// SIMATIC S7-200 project (STEP 7-Micro/WIN), CPU 224 REL 02.00

SYMBOL_TABLE Panel
LimInf_FallaCad  VD1920   // Limite inferior para falla sincronización de cadena
LimSup_FallaCad  VD1930   // Limite superior para falla sincronización de cadena
Time_Pusher_Fuera_Pos T105     // Timer, pusher fuera de posición
dAux40           VD2040   // DWAux40
dAux30           VD2030   // DWAux30
dAux20           VD2020   // DWAux20
dwAuxAlaPre      VD2004   // Aux de Alarma Presente
dwAuxMem         VD2002   // Aux Mem de Alarmas
dwAux3           VD2006   // AuxRecAlarmas
WFallas          VW100    // Para Panel_Word de Fallas en el programa
Panel_Habilitador V100.0   // Para Panel_Mark Habilitador de secuencia
Panel_Parada_Emergen V100.1   // Para Panel_Mark Parada de Emergencia (Puertas, pulsador)
Panel_Termicas1  V100.2   // Para Panel_Mark Termicas1 (Mot.Ppal, Bba Vacio, Hotmelt)
Panel_Termicas2  V100.3   // Para Panel_Mark  Termicas2 (Brazo, Pusher, Cinta Transporta.)
Panel_Cadena_Ppal V100.4   // Para Panel_Mark Seguridad Cadena principal Cortada
Panel_NO_Hay_Cajas V100.5   // Para Panel_Mark No Hay Cajas en el Cargador
Panel_Falla_MotorPusher V100.6   // Para Panel_Falla Motor Pusher
Panel_Falla_SsrPusher V100.7   // Para Panel_Falla Piston Pusher
Panel_Hotmelt_No_listo V101.0   // Para Panel_Mark Hotmelt No listo (señal externa)
Panel_Hotmelt_OFF V101.1   // Para Panel_Mark Hotmelt OFF
Panel_Cajas_Trabadas V101.2   // Para Panel_Mark Cajas Trabadas
Panel_Solapa_Trasea V101.3   // Para Panel_Mark Solapa Trasera abierta
Panel_Tiem_Sin_Hotmelt V101.4   // Para Panel_Falla por tiempo transcurrido sin Hotmelt OK
Panel_Solapa_Abierta V101.5   // Para Panel_SOLAPA TRASERA ABIERTA
Panel_Caja_Trabada_Sali V101.6   // Para Panel_CAJA NO SALIÓ DE LA MÁQUINA
Panel_FallaCajaCaida V101.7   // Para Panel_Falla caja cerrada en cadena
Panel_Falla_1SnsPucher V1836.0  // Falla Falto Confirmacion de 1 Sns del lo extremos Pusher
Panel_Falla_SsrEncDes V1836.1  // Falla SENSOR ENCOLADO DESENFOCADO
Panel_Falla_CadenaDesi V1836.2  // Falla CADENA DESINCRONIZADA
Panel_Falla_Push_Fuera V1836.3  // Falla PUSHER FUERA DE POSICION
Panel_Fall_Res_1836_4 V1836.4
Panel_Fall_Res_1836_5 V1836.5
Panel_Fall_Res_1836_6 V1836.6
Panel_Fall_Res_1836_7 V1836.7
Panel_Fall_Res_1837_0 V1837.0
Panel_Fall_Res_1837_1 V1837.1
Panel_Fall_Res_1837_2 V1837.2
Panel_Fall_Res_1837_3 V1837.3
Panel_Fall_Res_1837_4 V1837.4
Panel_Fall_Res_1837_5 V1837.5
Panel_Fall_Res_1837_6 V1837.6
Panel_Fall_Res_1837_7 V1837.7
Mem_Habilitador  V1820.0  // Memorizadas_Mark Habilitador de secuencia
Mem_Parada_Emergen V1820.1  // Memorizadas_Mark Parada de Emergencia (Puertas, pulsador)
Mem_Trmicas1     V1820.2  // Memorizadas_Mark Termicas1 (Mot.Ppal, Bba Vacio, Hotmelt)
Mem_Termicas2    V1820.3  // Memorizadas_Mark  Termicas2 (Brazo, Pusher, Cinta Transporta.)
Mem_Cadena_Ppal  V1820.4  // Memorizadas_Mark Seguridad Cadena principal Cortada
Mem_NO_Hay_Cajas V1820.5  // Memorizadas_Mark No Hay Cajas en el Cargador
Mem_Falla_MotPusher V1820.6  // Memorizadas_Falla Motor Pusher
Mem_Falla_PistPusher V1820.7  // Memorizadas_Falla Piston Pusher
Mem_Hotmelt_No_listo V1821.0  // Memorizadas_Mark Hotmelt No listo (señal externa)
Mem_Hotmelt_OFF  V1821.1  // Memorizadas_Mark Hotmelt OFF
Mem_Cajas_Trabadas V1821.2  // Memorizadas_Mark Cajas Trabadas
Mem_Solapa_Trasea V1821.3  // Memorizadas_Mark Solapa Trasera abierta
Mem_Tiem_Sin_Hotmelt V1821.4  // Memorizadas_Falla por tiempo transcurrido sin Hotmelt OK
Mem_Reserv_101_5 V1821.5  // Memorizadas_v1821.5 RESERVA
Mem_Reserv_101_6 V1821.6  // Memorizadas_v1821.6 RESERVA
Mem_Reserv_101_7 V1821.7  // Memorizadas_v1821.7 RESERVA
Tiempo_Encolado_1 VW102    // Word de tiempo para ENCOLADO 1º Solapa
Tiempo_Encolado_2 VW104    // Word de tiempo para ENCOLADO 2º Solapa
Tiempo_NO_Encolar VW106    // Word de tiempo para NO ENCOLADO
Panel_Timer_Corte_Vacio VW108    // De Panel_Word de tiempo para cortar VACIO
Panel_Sel_Caja   VW110    // De Panel Selección de Programa por Tipo de Caja
Valor_Encoder_ParaPanel VD120    // Valor Actual del Encoder al Panel
Byte_Motor_Ppal_Panel MB5      // Byte para dar marcha al motor Ppal desde el Panel
Marcha_Motor_Ppal_Panel M5.0     // Mark para dar marcha al motor Ppal desde el Panel
Panel_Tie_Enc_1_0 VW160    // Tiempo Encolado 1º Solapa Caja 15x1000
Panel_Tie_Enc_2_0 VW162    // Tiempo Encolado 2º Solapa Caja 15x1000
Panel_Tie_NoEnc_0 VW164    // Tiempo No Encolado Caja 15x1000
Panel_Tie_Enc_1_1 VW166    // Tiempo Encolado 1º Solapa Caja 12x1500
Panel_Tie_Enc_2_1 VW168    // Tiempo Encolado 2º Solapa Caja 12x1500
Panel_Tie_NoEnc_1 VW170    // Tiempo No Encolado Caja 12x1500
Panel_Tie_Enc_1_2 VW172    // Tiempo Encolado 1º Solapa Caja 12x1000
Panel_Tie_Enc_2_2 VW174    // Tiempo Encolado 2º Solapa Caja 12x1000
Panel_Tie_NoEnc_2 VW176    // Tiempo No Encolado Caja 12x1000
Panel_Tie_Enc_1_3 VW178    // Tiempo Encolado 1º Solapa Caja 12x750
Panel_Tie_Enc_2_3 VW180    // Tiempo Encolado 2º Solapa Caja 12x750
Panel_Tie_NoEnc_3 VW182    // Tiempo No Encolado Caja 12x750
Hab_Falla_18362  M29.2    // Hab_Falla_Sic_Cadena
END_SYMBOL_TABLE

SYMBOL_TABLE I/O
iEncoder_Fase_A  I0.0     // Encoder pulso A
iEncoder_Fase_B  I0.1     // Encoder pulso B
iEncoder_Cero    I0.2     // Encoder pulso 0
iSsr_Area_Encolado I0.3     // Sensor Caja en Area Encolado
iSelect_Auto     I0.4     // Selectora en  automatico
iSelect_Test     I0.5     // Selectora en  Test
iSsr_Brazo_BielaLarga I0.6     // Sensor Brazo biela larga
iSsr_Brazo_BielaCorta I0.7     // Sensor Brazo biela corta
iHotmelt_Ready   I1.0     // Hotmelt Ready
iSel_arr_dir_var I1.1     // Selectora arranque motor directo o con variador
iSsr_CajaCaida   I1.2     // Sensor de caja no abierta/caida en cadena
i1_3             I1.3     // Reserva
iSsr_Pusher_Atras I1.4     // Pusher atras Brazo completo habilitador de secuencia
iHabilitador_Linea_ext I1.5     // Habilitador externo Linea de salida
iSsr_Cajas_Cargador I3.0     // Sensor Presencia de Cajas en Cargador
iHotmelt_ON      I3.1     // Contacto Hotmelt ON
iPton_Pusher_Atras I3.2     // Sensor Piston de Pusher Atrás
iPton_Pusher_Adelante I3.3     // Sensor Piston de Pusher Adelante
iSsr_Caja_Trabada_Out I3.4     // Sensor Caja Trabada a la Salida
iSsr_Cadena_Cortada I3.5     // Seguridad cadena cortada
iSsr_Linea_Llena I3.6     // Sensor de Linea Llena
iSsr_Solapa_Trasera I3.7     // Sensor Solapa trasera abierta
iHabilitador     I2.0     // Habilitador
iParada_Emergencia I2.1     // Parada de emergencia
iReset_Fallas    I2.2     // Reset de Fallas
iCadena_Termicas_1 I2.3     // Cadena de termicas motores pricipal,bba vacio, hotmelt
iCadena_Termicas_2 I2.4     // Cadena de termicas motores brazo, presionador, tranportadora
iMarcha          I2.5     // Start
iParada          I2.6     // Stop
iBrazo_Up_Down   I2.7     // Brazo arriba/abajo
oMotor_Ppal      Q0.0     // K_Motor principal
oBba_Vacio       Q0.1     // K_Bba vacio
oMotor_Brazo     Q0.2     // K_Brazo
oMotor_Pusher    Q0.3     // K_Pusher
oMotor_Cinta_Transport Q0.4     // K_Transportadora
oLuz_Roja        Q0.5     // Luz Roja
oLuz_Marcha      Q0.6     // Luz Verde
oAlimenta_Cadena_Emer Q0.7     // Salida a Linea de emergencia
oPiston_Cargador_Cajas Q1.0     // Piston Cargador de Cajas
oPiston_Separad_Cajas Q1.1     // Piston Separadores de Cajas
oActivar_Vacio   Q2.0     // Electrovalvula  Activar Vacio
oCerrar_Brzo_Sost_Cajas Q2.1     // Electrovalvula  Cerrar brasitos sostenedores de caja al inicio
oCerrar_Solapa_Trasera Q2.2     // Electrovalvula  Cerrar solapa trasera
oSostener_P_Escuadrar Q2.3     // Electrovalvula  Sostener caja para escuadrar
oActivar_Hotmelt Q2.4     // Electrovalvula  Activar salida de Hotmelt
oActivar_Piston_Pusher Q2.5     // Electrovalvula  Activar Piston de Pusher
oCerrar_Solapas_Armado Q2.6     // Electrovalvula  Cerrar solapas Traseras en area de Armado
oActiv_Escuadrador Q2.7     // Electrovalvula  Activar Pistones para Escuadrar
oMotor_Brazo_Var Q3.0     // Arranque con variador del brazo
o3_1             Q3.1     // No anda
oFreno_Brazo     Q3.2     // Freno Motor Brazo
o3_3             Q3.3     // Libre
o3_4             Q3.4     // Libre
o3_5             Q3.5     // Libre
o3_6             Q3.6     // Libre
o3_7             Q3.7     // Libre
END_SYMBOL_TABLE

SYMBOL_TABLE Motores
Estado_Motores   MB10     // Byte de estado de los motores
Marcha_Mot_Princ M10.0    // Mark Marcha Motor Principal
Marcha_Bba_Vacio M10.1    // Mark Marcha Bomba de vacio
Marcha_Brazo_Succ M10.2    // Mark Marcha Brazo Succionador
Marcha_Pusher    M10.3    // Mark Marcha Pusher
Marcha_Cinta_Transp M10.4    // Mark Marcha Cinta Transportadora
Reserva          M10.5    // Reserva
Reserva1         M10.6    // Reserva
Reserva2         M10.7    // Reserva
END_SYMBOL_TABLE

SYMBOL_TABLE Seguridad Fallas
Estado_Seguridad MB20     // Estado del byte de seguridad
Habilitador      M20.0    // Mark Habilitador de secuencia
Parada_Emergencia M20.1    // Mark Parada de Emergencia (Puertas, pulsador)
Termicas_1       M20.2    // Mark Termicas1 (Mot.Ppal, Bba Vacio, Hotmelt)
Termicas_2       M20.3    // Mark  Termicas2 (Brazo, Pusher, Cinta Transporta.)
Cadena_Ppal      M20.4    // Mark Seguridad Cadena principal
Res1             M20.5    // Reserva
Res2             M20.6    // Reserva
Res3             M20.7    // Reserva
Falla_Gral       M21.0    // Mark de Falla General para mandar todo a Reposo
Hotmelt_OK       M21.1    // Mark de Hotmel OK
Parada_Espera    M21.2    // Parada Ordenada o Espera por Equipos listos
END_SYMBOL_TABLE

SYMBOL_TABLE Símbolos S7-200
Bit1             SM0.0    // Siempre ON
CicIni           SM0.1    // ON sólo en el primer ciclo
Reloj_1s         SM0.5    // Reloj ON durante 0,5 s, OFF durante 0,5 s, tiempo de ciclo = 1 s.
Actualizar_CV_HSC0 SM37.6   // Actualizar el valor actual de HSC0: 0=no actualizar; 1=actualizar
Control_HSC0     SMB37    // Configurar y controlar HSC0
CV_HSC0          SMD38    // Nuevo valor actual de HSC0
PV_HSC0          SMD42    // Nuevo valor predeterminado de HSC0
END_SYMBOL_TABLE

SYMBOL_TABLE Luces y Externas
Estado_Varios    MB15     // Byte Estado de varios
Luz_Roja         M15.0    // Indicacion Luz Roja
Luz_Verde        M15.1    // Indicacion Luz Verde
Salida_Emergencia M15.2    // Mark de Salida para Línea de emergencia
Reserv1          M15.3    // Reserva
Reserv2          M15.4    // Reserva
Hotmelt_ON       M15.5    // Mark Hotmelt ON
Hotmelt_Listo    M15.6    // Mark Hotmelt Listo (Señal Externa)
Linea_Salida_Habilitada M15.7    // Mark Habilitador Externo linea de salida
END_SYMBOL_TABLE

SYMBOL_TABLE Válvulas
Estado_Valvulas  MW12     // Estado de las Válvulas
Activar_Vacio    M12.0    // Mark Activar Vacio
Cerrar_Solapas_Armado M12.1    // Mark Cerrar solapas Traseras en area de Armado
Cerrar_Solapa_Trasera M12.2    // Mark Cerrar solapa trasera
Activ_Escuadrador M12.3    // Mark Activar Pistones para Escuadrar
Activar_Hotmelt  M12.4    // Mark Activar salida de Hotmelt
Activar_Piston_Pusher M12.5    // Mark Activar Piston de Pusher
Cerrar_Brzo_Sost_Cajas M12.6    // Mark Cerrar brasitos sostenedores de caja al inicio
Sostener_P_Escuadrar M12.7    // Mark Sostener caja para escuadrar
Piston_Cargador_Cajas M13.0    // Mark Activar Piston del cargador cajas
Piston_Separad_Cajas M13.1    // Mark Activar Pistonnes separadores de cajas
Reser1           M13.2    // Reserva
Reser2           M13.3    // Reserva
Reser3           M13.4    // Reserva
Reser4           M13.5    // Reserva
Reser5           M13.6    // Reserva
Reser6           M13.7    // Reserva
END_SYMBOL_TABLE

SYMBOL_TABLE Selectoras_Pulsa
Est_Selectoras_Pulsad MB22     // Estado de las Selectoras y de los Pulsadores
Pulsador_Reset_Fallas M22.0    // Mark Pulsador Reset de Problemas
Pulsador_Start   M22.1    // Mark Pulsador Start
Pulsador_Stop    M22.2    // Mark Pulsador Stop
Pulsador_Brazo_Up_D M22.3    // Mark Pulsador Brazo Arriba / Abajo
Selectora_Auto   M22.4    // Mark Selectora en Auto
Selectora_Test   M22.5    // Mark Selectora en Test
Reserva_1        M22.6    // Brazo Subió o está bajando
Reserva_2        M22.7    // Reserva
END_SYMBOL_TABLE

SYMBOL_TABLE Sensores
Sensores         MW24     // Word Estado de los sensores
Ssr_Caja_Area_Pegado M24.0    // Mark Sensor Detector de Caja para Pegar
Ssr_Brazo_Abajo  M24.1    // Mark Sensor Brazo Abajo (biela larga) para vacio
Ssr_Brazo_Bajando M24.2    // Mark Sensor Brazo Arriba (biela corta) para vacio
Ssr_Linea_Llena  M24.3    // Mark Sensor de Linea Llena
Ssr_Pist_Pusher_Atras M24.4    // Mark Sensor de Piston del Pusher Atras
Ssr_Pist_Pusher_Adelant M24.5    // Mark Sensor de Piston del Pusher Adelante
Ssr_Caja_Trabada_Out M24.6    // Mark Sensor de cajas Trabadas a la salida
Ssr_Falta_Caja_Cargador M24.7    // Mark Sensor Falta de cajas en el Cargador
Ssr_Slpa_Tras_Abiert M25.0    // Mark Sensor Solapa trasera abierta
Ssr_Pusher_Atras M25.1    // Mark Sensor de Pusher Atras
Ssr_Hay_Caja_Cargador M25.2    // Mark Sensor Presencia de cajas en el Cargador
Res_2            M25.3    // Reserva
Res_3            M25.4    // Reserva
Res_4            M25.5    // Reserva
Res_5            M25.6    // Reserva
Res_6            M25.7    // Reserva
END_SYMBOL_TABLE

SYMBOL_TABLE Estado_Variables
_1sD1            VD0      // Valor del estado 1 actual (por cada bit 1 estado)
_1sW1            VW0
_1s0             V0.0     // S1_Estado0
_1s1             V0.1     // S1_Estado1 Reposo
_1s2             V0.2     // S1_Estado2 Inicio
_1s3             V0.3     // S1_Estado3 Activo Bba Vacio
_1s4             V0.4     // S1_Estado4 Activo cinta transp. y motor Ppal
_1s5             V0.5     // S1_Estado5 Encolar 1º solapa
_1s6             V0.6     // S1_Estado6 Espera
_1s7             V0.7     // S1_Estado7 Encolar 2º Solapa
_1s8             V1.0     // S1_Estado8 Espera
_1s9             V1.1     // S1_Estado9 Activo secuencia 2 y 3
_1s10            V1.2     // S1_Estado10 Activo secuencia 2 y 3
_1s11            V1.3     // S1_Estado11 Caja mal Armada
_1s12            V1.4     // S1_Estado12 Sin Cajas
_1s13            V1.5     // S1_Estado13 Reconocer Fallas
_1s14            V1.6     // S1_Estado14 Falla Pusher
_1s15            V1.7     // S1_Estado15
_1s16            V2.0     // S1_Estado16
_1s17            V2.1     // S1_Estado17
_1s18            V2.2     // S1_Estado18
_1s19            V2.3     // S1_Estado19
_1s20            V2.4     // S1_Estado20
_1s21            V2.5     // S1_Estado21
_1s22            V2.6     // S1_Estado22
_1s23            V2.7     // S1_Estado23
_1s24            V3.0     // S1_Estado24
_1s25            V3.1     // S1_Estado25
_1s26            V3.2     // S1_Estado26
_1s27            V3.3     // S1_Estado27
_1s28            V3.4     // S1_Estado28
_1s29            V3.5     // S1_Estado29
_1s30            V3.6     // S1_Estado30
_1s31            V3.7     // S1_Estado31
_2sw1            VW4      // Valor del estado 2 actual (por cada bit 1 estado)
_2s0             V4.0     // S2_Estado0
_2s1             V4.1     // S2_Estado1 Reposo
_2s2             V4.2     // S2_Estado2 Inicio
_2s3             V4.3     // S2_Estado3 Esscuadrar y cerrar solapas traseras
_2s4             V4.4     // S2_Estado4 Cerrar solapas sin pegamento
_2s5             V4.5     // S2_Estado5 Marcha motor Pusher
_2s6             V4.6     // S2_Estado6 Entrar piston Pusher
_2s7             V4.7     // S2_Estado7 Sacar Piston Pusher
_2s8             V5.0     // S2_Estado8 Fin Armado
_2s9             V5.1     // S2_Estado9 Falla Psuher
_2s10            V5.2     // S2_Estado10
_2s11            V5.3     // S2_Estado11
_2s12            V5.4     // S2_Estado12
_2s13            V5.5     // S2_Estado13
_2s14            V5.6     // S2_Estado14
_2s15            V5.7     // S2_Estado15
_3sw1            VW6      // Valor del estado 3 actual (por cada bit 1 estado)
_3s0             V6.0     // S3_Estado0
_3s1             V6.1     // S3_Estado1 Reposo
_3s2             V6.2     // S3_Estado2 Marchar Motor Brazo
_3s3             V6.3     // S3_Estado3 Activar Vacio
_3s4             V6.4     // S3_Estado4 Cortar Vacio
_3s5             V6.5     // S3_Estado5 Detener Motor Brazo
_3s6             V6.6     // S3_Estado6
_3s7             V6.7     // S3_Estado7
_3s8             V7.0     // S3_Estado8
_3s9             V7.1     // S3_Estado9
_3s10            V7.2     // S3_Estado10
_3s11            V7.3     // S3_Estado11
_3s12            V7.4     // S3_Estado12
_3s13            V7.5     // S3_Estado13
_3s14            V7.6     // S3_Estado14
_3s15            V7.7     // S3_Estado15
_4sw1            VW8      // Valor del estado 4 actual (por cada bit 1 estado)
_4s0             V8.0     // S4_Estado0
_4s1             V8.1     // S4_Estado1 Reposo
_4s2             V8.2     // S4_Estado2 Activación Pistón Cargador
_4s3             V8.3     // S3_Estado3 Desactivación Pistón Cargador
_4s4             V8.4     // S3_Estado4 Falla por Falta de Cajas
_4s5             V8.5     // S4_Estado5
_4s6             V8.6     // S4_Estado6
_4s7             V8.7     // S4_Estado7
_4s8             V9.0     // S4_Estado8
_4s9             V9.1     // S4_Estado9
_4s10            V9.2     // S4_Estado10
_4s11            V9.3     // S4_Estado11
_4s12            V9.4     // S4_Estado12
_4s13            V9.5     // S4_Estado13
_4s14            V9.6     // S4_Estado14
_4s15            V9.7     // S4_Estado15
END_SYMBOL_TABLE

SYMBOL_TABLE Timers y Contadores
Time_Ssr_Enc_Desen T104     // Timer, de Sns de Encolado desenfocado
Time_Fin_Escuadre T33      // TON_10 Timer Tiempo de Escuadre
Time_Inicio_Pusher T34      // TON_10 Timer Tiempo de Retardo de Pusher
Time_Encolado_1  T35      // TON_10 Timer Tiempo Encolado 1º Solapa
Time_NO_Encolado T36      // TON_10 Timer Tiempo NO Encolado
Time_Falta_Caja_Cargad T37      // TON_100 Timer Tiempo Detección Falta de Cajas Cargador
Time_Arranque_Bba T38      // TON_100 Timer Tiempo Arranque Bomba Vacio
Time_Arranque_CyMPpal T39      // TON_100 Timer Tiempo Arranque Cinta y Motor Ppal.
Time_Falla_Pusher T40      // TON_100 Timer Tiempo Falla Motor Pusher
Time_Falla_PistonPusher T41      // TON_100 Timer Tiempo Falla Piston Pusher
Time_Hay_Caja_Cargador T42      // TON_100 Timer Tiempo Detección Presencia Cajas Cargador
Time_Act_Carg_Caja T43      // TON_100 Timer Activación Pistón Cargador de Cajas
Time_Desact_Carg_Caja T44      // TON_100 Timer Desactivación Pistón Cargador de Cajas
Time_Desact_Solapas T45      // TON_100 Timer Desactivación Solapas Armado
Time_Espera_DetCarg T46      // TON_100 Timer Espera luego de detener cargador de cajas
TON_Reset        T47      // Timer 5 segundos con Reset de Alarmas
Time_Encolado_2  T97      // TON_10 Timer Tiempo Encolado 2º Solapa
Time_Corte_Vacio T100     // TON_10 Timer Retardo corte Vacio, Brazo Bajando
Time_SsrLineaLlena T101     // TON_100 Timer Ssr Linea Llena
Time_Falla_Hotmelt T102     // TOF_100 Timer para parar por Falla en Equipo Hotmelt
Time_Out_SinCajas T103
D_Pnel_T_Escuadre VW130    // Panel_TON_10 Timer Tiempo de Escuadre
D_Pnel_T_RetardoPushe VW132    // Panel_TON_10 Timer Tiempo de Retardo de Pusher
D_Pnel_T_Arranque_Bba VW134    // Panel_TON_100 Timer Tiempo Arranque Bomba Vacio
D_Pnel_T_ArranqCyMPpal VW136    // Panel_TON_100 Timer Tiempo Arranque Cinta y Motor Ppal.
D_Pnel_T_Falla_Pusher VW138    // Panel_TON_100 Timer Tiempo Falla Motor Pusher
D_Pnel_T_FallaPistPush VW140    // Panel_TON_100 Timer Tiempo Falla Piston Pusher
CTD_Alim_Cajas   C1       // Contador de Intentos de Alimentador de Cajas
END_SYMBOL_TABLE

SYMBOL_TABLE Standart Panel
TcSis8           V1862.0  // Sin Uso
Del_Ins          V1862.1  // Tecla Del/Ins
HrdCopy          V1862.2  // Tecla Hard Copy
Shift            V1862.3  // Tecla Shift
DecPt            V1862.4  // Tecla punto decimal
TcMasmenos       V1862.5  // Tecla +/-
TcSis14          V1862.6  // Sin Uso
TcSis15          V1862.7  // Sin Uso
Info             V1863.0  // Tecla Info
AlAck            V1863.1  // Tecla reconocimiento de alarmas
TcSis2           V1863.2  // Sin Uso
Esc              V1863.3  // Tecla escape
TcSis4           V1863.4  // Sin Uso
TcSis5           V1863.5  // Sin Uso
Enter            V1863.6  // Tecla Enter
TcSis7           V1863.7  // Sin Uso
Num8             V1864.0  // Tecla numero 8
Num9             V1864.1  // Tecla numero 9
TcSis26          V1864.2  // Sin Uso
TcSis27          V1864.3  // Sin Uso
TcSis28          V1864.4  // Sin Uso
TcSis29          V1864.5  // Sin Uso
TcSis30          V1864.6  // Sin Uso
TcGrp            V1864.7  // Grupo teclas de sistema
Num0             V1865.0  // Tecla numero 0
Num1             V1865.1  // Tecla numero 1
Num2             V1865.2  // Tecla numero 2
Num3             V1865.3  // Tecla numero 3
Num4             V1865.4  // Tecla numero 4
Num5             V1865.5  // Tecla numero 5
Num6             V1865.6  // Tecla numero 6
Num7             V1865.7  // Tecla numero 7
Opf9             V1866.0  // OP,tecla de funcion 9
Opf10            V1866.1  // OP,tecla de funcion 10
Opf11            V1866.2  // OP,tecla de funcion 11
Opf12            V1866.3  // OP,tecla de funcion 12
Opf13            V1866.4  // OP,tecla de funcion 13
Opf14            V1866.5  // OP,tecla de funcion 14
Opf15            V1866.6  // OP,tecla de funcion 15
Opf16            V1866.7  // OP,tecla de funcion 16
Opf1             V1867.0  // OP,tecla de funcion 1
Opf2             V1867.1  // OP,tecla de funcion 2
Opf3             V1867.2  // OP,tecla de funcion 3
Opf4             V1867.3  // OP,tecla de funcion 4
Opf5             V1867.4  // OP,tecla de funcion 5
Opf6             V1867.5  // OP,tecla de funcion 6
Opf7             V1867.6  // OP,tecla de funcion 7
Opf8             V1867.7  // OP,tecla de funcion 8
MesSigCmp4       V1868.0  // OP, activacion de bit, desplazamiento 24
MesAntCmp4       V1868.1  // OP, activacion de bit, desplazamiento 25
MesSigCmp5       V1868.2  // OP, activacion de bit, desplazamiento 26
MesAntCmp5       V1868.3  // OP, activacion de bit, desplazamiento 27
MesSigCmp6       V1868.4  // OP, activacion de bit, desplazamiento 28
MesAntCmp6       V1868.5  // OP, activacion de bit, desplazamiento 29
Act30            V1868.6  // OP, activacion de bit, desplazamiento 30
Act31            V1868.7  // OP, activacion de bit, desplazamiento 31
PuHabCmp         V1869.0  // Pulsador para habilitar compresores
PuInhCmp         V1869.1  // Pulsador para inhabilitar compresores
MesSigCmp1       V1869.2  // OP, activacion de bit, desplazamiento 18
MesAntCmp1       V1869.3  // OP, activacion de bit, desplazamiento 19
MesSigCmp2       V1869.4  // OP, activacion de bit, desplazamiento 20
MesAntCmp2       V1869.5  // OP, activacion de bit, desplazamiento 21
MesSigCmp3       V1869.6  // OP, activacion de bit, desplazamiento 22
MesAntCmp3       V1869.7  // OP, activacion de bit, desplazamiento 23
Act40            V1870.0  // OP, activacion de bit, desplazamiento 40
Act41            V1870.1  // OP, activacion de bit, desplazamiento 41
Act42            V1870.2  // OP, activacion de bit, desplazamiento 42
Act43            V1870.3  // OP, activacion de bit, desplazamiento 43
Act44            V1870.4  // OP, activacion de bit, desplazamiento 44
Act45            V1870.5  // OP, activacion de bit, desplazamiento 45
Act46            V1870.6  // OP, activacion de bit, desplazamiento 46
Act47            V1870.7  // OP, activacion de bit, desplazamiento 47
Act32            V1871.0  // OP, activacion de bit, desplazamiento 32
Act33            V1871.1  // OP, activacion de bit, desplazamiento 33
Act34            V1871.2  // OP, activacion de bit, desplazamiento 34
Act35            V1871.3  // OP, activacion de bit, desplazamiento 35
Act36            V1871.4  // OP, activacion de bit, desplazamiento 36
Act37            V1871.5  // OP, activacion de bit, desplazamiento 37
Act38            V1871.6  // OP, activacion de bit, desplazamiento 38
Act39            V1871.7  // OP, activacion de bit, desplazamiento 39
Act56            V1872.0  // OP, activacion de bit, desplazamiento 56
Act57            V1872.1  // OP, activacion de bit, desplazamiento 57
Act58            V1872.2  // OP, activacion de bit, desplazamiento 58
Act59            V1872.3  // OP, activacion de bit, desplazamiento 59
Act60            V1872.4  // OP, activacion de bit, desplazamiento 60
Act61            V1872.5  // OP, activacion de bit, desplazamiento 61
Act62            V1872.6  // OP, activacion de bit, desplazamiento 62
Act63            V1872.7  // OP, activacion de bit, desplazamiento 63
Act48            V1873.0  // OP, activacion de bit, desplazamiento 48
Act49            V1873.1  // OP, activacion de bit, desplazamiento 49
Act50            V1873.2  // OP, activacion de bit, desplazamiento 50
Act51            V1873.3  // OP, activacion de bit, desplazamiento 51
Act52            V1873.4  // OP, activacion de bit, desplazamiento 52
Act53            V1873.5  // OP, activacion de bit, desplazamiento 53
Act54            V1873.6  // OP, activacion de bit, desplazamiento 54
Act55            V1873.7  // OP, activacion de bit, desplazamiento 55
fTcSis8          V1894.0  // Sin Uso
fDel_Ins         V1894.1  // Tecla Del/Ins
fHrdCopy         V1894.2  // Tecla Hard Copy
fShift           V1894.3  // Tecla Shift
fDecPt           V1894.4  // Tecla punto decimal
fTcMasmenos      V1894.5  // Tecla +/-
fTcSis14         V1894.6  // Sin Uso
fTcSis15         V1894.7  // Sin Uso
fInfo            V1895.0  // Tecla Info
fAlAck           V1895.1  // Tecla reconocimiento de alarmas
fTcSis2          V1895.2  // Sin Uso
fEsc             V1895.3  // Tecla escape
fTcSis4          V1895.4  // Sin Uso
fTcSis5          V1895.5  // Sin Uso
fEnter           V1895.6  // Tecla Enter
fTcSis7          V1895.7  // Sin Uso
fNum8            V1896.0  // Tecla numero 8
fNum9            V1896.1  // Tecla numero 9
fTcSis26         V1896.2  // Sin Uso
fTcSis27         V1896.3  // Sin Uso
fTcSis28         V1896.4  // Sin Uso
fTcSis29         V1896.5  // Sin Uso
fTcSis30         V1896.6  // Sin Uso
fTcGrp           V1896.7  // Grupo teclas de sistema
fNum0            V1897.0  // Tecla numero 0
fNum1            V1897.1  // Tecla numero 1
fNum2            V1897.2  // Tecla numero 2
fNum3            V1897.3  // Tecla numero 3
fNum4            V1897.4  // Tecla numero 4
fNum5            V1897.5  // Tecla numero 5
fNum6            V1897.6  // Tecla numero 6
fNum7            V1897.7  // Tecla numero 7
fOpf9            V1898.0  // Flanco OP,tecla de funcion 9
fOpf10           V1898.1  // Flanco OP,tecla de funcion 10
fOpf11           V1898.2  // Flanco OP,tecla de funcion 11
fOpf12           V1898.3  // Flanco OP,tecla de funcion 12
fOpf13           V1898.4  // Flanco OP,tecla de funcion 13
fOpf14           V1898.5  // Flanco OP,tecla de funcion 14
fOpf15           V1898.6  // Flanco OP,tecla de funcion 15
fOpf16           V1898.7  // Flanco OP,tecla de funcion 16
fOpf1            V1899.0  // Flanco OP,tecla de funcion 1
fOpf2            V1899.1  // Flanco OP,tecla de funcion 2
fOpf3            V1899.2  // Flanco OP,tecla de funcion 3
fOpf4            V1899.3  // Flanco OP,tecla de funcion 4
fOpf5            V1899.4  // Flanco OP,tecla de funcion 5
fOpf6            V1899.5  // Flanco OP,tecla de funcion 6
fOpf7            V1899.6  // Flanco OP,tecla de funcion 7
fOpf8            V1899.7  // Flanco OP,tecla de funcion 8
fMesSigCmp4      V1900.0  // Flanco OP, activacion de bit, desplazamiento 24
fMesAntCmp4      V1900.1  // Flanco OP, activacion de bit, desplazamiento 25
fMesSigCmp5      V1900.2  // Flanco OP, activacion de bit, desplazamiento 26
fMesAntCmp5      V1900.3  // Flanco OP, activacion de bit, desplazamiento 27
fMesSigCmp6      V1900.4  // Flanco OP, activacion de bit, desplazamiento 28
fMesAntCmp6      V1900.5  // Flanco OP, activacion de bit, desplazamiento 29
fAct30           V1900.6  // Flanco OP, activacion de bit, desplazamiento 30
fAct31           V1900.7  // Flanco OP, activacion de bit, desplazamiento 31
fPuHabCmp        V1901.0  // Flanco Pulsador para habilitar compresores
fPuInhCmp        V1901.1  // Flanco Pulsador para inhabilitar compresores
fMesSigCmp1      V1901.2  // Flanco OP, activacion de bit, desplazamiento 18
fMesAntCmp1      V1901.3  // Flanco OP, activacion de bit, desplazamiento 19
fMesSigCmp2      V1901.4  // Flanco OP, activacion de bit, desplazamiento 20
fMesAntCmp2      V1901.5  // Flanco OP, activacion de bit, desplazamiento 21
fMesSigCmp3      V1901.6  // Flanco OP, activacion de bit, desplazamiento 22
fMesAntCmp3      V1901.7  // Flanco OP, activacion de bit, desplazamiento 23
fAct40           V1902.0  // Flanco OP, activacion de bit, desplazamiento 40
fAct41           V1902.1  // Flanco OP, activacion de bit, desplazamiento 41
fAct42           V1902.2  // Flanco OP, activacion de bit, desplazamiento 42
fAct43           V1902.3  // Flanco OP, activacion de bit, desplazamiento 43
fAct44           V1902.4  // Flanco OP, activacion de bit, desplazamiento 44
fAct45           V1902.5  // Flanco OP, activacion de bit, desplazamiento 45
fAct46           V1902.6  // Flanco OP, activacion de bit, desplazamiento 46
fAct47           V1902.7  // Flanco OP, activacion de bit, desplazamiento 47
fAct32           V1903.0  // Flanco OP, activacion de bit, desplazamiento 32
fAct33           V1903.1  // Flanco OP, activacion de bit, desplazamiento 33
fAct34           V1903.2  // Flanco OP, activacion de bit, desplazamiento 34
fAct35           V1903.3  // Flanco OP, activacion de bit, desplazamiento 35
fAct36           V1903.4  // Flanco OP, activacion de bit, desplazamiento 36
fAct37           V1903.5  // Flanco OP, activacion de bit, desplazamiento 37
fAct38           V1903.6  // Flanco OP, activacion de bit, desplazamiento 38
fAct39           V1903.7  // Flanco OP, activacion de bit, desplazamiento 39
fAct56           V1904.0  // Flanco OP, activacion de bit, desplazamiento 56
fAct57           V1904.1  // Flanco OP, activacion de bit, desplazamiento 57
fAct58           V1904.2  // Flanco OP, activacion de bit, desplazamiento 58
fAct59           V1904.3  // Flanco OP, activacion de bit, desplazamiento 59
fAct60           V1904.4  // Flanco OP, activacion de bit, desplazamiento 60
fAct61           V1904.5  // Flanco OP, activacion de bit, desplazamiento 61
fAct62           V1904.6  // Flanco OP, activacion de bit, desplazamiento 62
fAct63           V1904.7  // Flanco OP, activacion de bit, desplazamiento 63
fAct48           V1905.0  // Flanco OP, activacion de bit, desplazamiento 48
fAct49           V1905.1  // Flanco OP, activacion de bit, desplazamiento 49
fAct50           V1905.2  // Flanco OP, activacion de bit, desplazamiento 50
fAct51           V1905.3  // Flanco OP, activacion de bit, desplazamiento 51
fAct52           V1905.4  // Flanco OP, activacion de bit, desplazamiento 52
fAct53           V1905.5  // Flanco OP, activacion de bit, desplazamiento 53
fAct54           V1905.6  // Flanco OP, activacion de bit, desplazamiento 54
fAct55           V1905.7  // Flanco OP, activacion de bit, desplazamiento 55
LedRoj9          V1996.0  // Led rojo permanente 9
LedRoj10         V1996.1  // Led rojo permanente 10
LedRoj11         V1996.2  // Led rojo permanente 11
LedRoj12         V1996.3  // Led rojo permanente 12
LedRoj13         V1996.4  // Led rojo permanente 13
LedRoj14         V1996.5  // Led rojo permanente 14
LedRoj15         V1996.6  // Led rojo permanente 15
LedRoj16         V1996.7  // Led rojo permanente 16
LedRoj1          V1997.0  // Led rojo permanente 1
LedRoj2          V1997.1  // Led rojo permanente 2
LedRoj3          V1997.2  // Led rojo permanente 3
LedRoj4          V1997.3  // Led rojo permanente 4
LedRoj5          V1997.4  // Led rojo permanente 5
LedRoj6          V1997.5  // Led rojo permanente 6
LedRoj7          V1997.6  // Led rojo permanente 7
LedRoj8          V1997.7  // Led rojo permanente 8
LedRojInt9       V1998.0  // Led rojo intermitente 9
LedRojInt10      V1998.1  // Led rojo intermitente 10
LedRojInt11      V1998.2  // Led rojo intermitente 11
LedRojInt12      V1998.3  // Led rojo intermitente 12
LedRojInt13      V1998.4  // Led rojo intermitente 13
LedRojInt14      V1998.5  // Led rojo intermitente 14
LedRojInt15      V1998.6  // Led rojo intermitente 15
LedRojInt16      V1998.7  // Led rojo intermitente 16
LedRojInt1       V1999.0  // Led rojo intermitente 1
LedRojInt2       V1999.1  // Led rojo intermitente 2
LedRojInt3       V1999.2  // Led rojo intermitente 3
LedRojInt4       V1999.3  // Led rojo intermitente 4
LedRojInt5       V1999.4  // Led rojo intermitente 5
LedRojInt6       V1999.5  // Led rojo intermitente 6
LedRojInt7       V1999.6  // Led rojo intermitente 7
LedRojInt8       V1999.7  // Led rojo intermitente 8
LedVer9          V2000.0  // Led verde permanente 9
LedVer10         V2000.1  // Led verde permanente 10
LedVer11         V2000.2  // Led verde permanente 11
LedVer12         V2000.3  // Led verde permanente 12
LedVer13         V2000.4  // Led verde permanente 13
LedVer14         V2000.5  // Led verde permanente 14
LedVer15         V2000.6  // Led verde permanente 15
LedVer16         V2000.7  // Led verde permanente 16
LedVer1          V2001.0  // Led verde permanente 1
LedVer2          V2001.1  // Led verde permanente 2
LedVer3          V2001.2  // Led verde permanente 3
LedVer4          V2001.3  // Led verde permanente 4
LedVer5          V2001.4  // Led verde permanente 5
LedVer6          V2001.5  // Led verde permanente 6
LedVer7          V2001.6  // Led verde permanente 7
LedVer8          V2001.7  // Led verde permanente 8
x9               V2002.0  // Marca auxiliar 9
x10              V2002.1  // Marca auxiliar 10
x11              V2002.2  // Marca auxiliar 11
x12              V2002.3  // Marca auxiliar 12
x13              V2002.4  // Marca auxiliar 13
x14              V2002.5  // Marca auxiliar 14
x15              V2002.6  // Marca auxiliar 15
x16              V2002.7  // Marca auxiliar 16
x1               V2003.0  // Marca auxiliar 1
x2               V2003.1  // Marca auxiliar 2
x3               V2003.2  // Marca auxiliar 3
x4               V2003.3  // Marca auxiliar 4
x5               V2003.4  // Marca auxiliar 5
x6               V2003.5  // Marca auxiliar 6
x7               V2003.6  // Marca auxiliar 7
x8               V2003.7  // Marca auxiliar 8
x25              V2004.0  // Marca auxiliar 25
x26              V2004.1  // Marca auxiliar 26
x27              V2004.2  // Marca auxiliar 27
x28              V2004.3  // Marca auxiliar 28
x29              V2004.4  // Marca auxiliar 29
x30              V2004.5  // Marca auxiliar 30
x31              V2004.6  // Marca auxiliar 31
x32              V2004.7  // Marca auxiliar 32
x17              V2005.0  // Marca auxiliar 17
x18              V2005.1  // Marca auxiliar 18
x19              V2005.2  // Marca auxiliar 19
x20              V2005.3  // Marca auxiliar 20
x21              V2005.4  // Marca auxiliar 21
x22              V2005.5  // Marca auxiliar 22
x23              V2005.6  // Marca auxiliar 23
x24              V2005.7  // Marca auxiliar 24
x41              V2006.0  // Marca auxiliar 41
x42              V2006.1  // Marca auxiliar 42
x43              V2006.2  // Marca auxiliar 43
x44              V2006.3  // Marca auxiliar 44
x45              V2006.4  // Marca auxiliar 45
x46              V2006.5  // Marca auxiliar 46
x47              V2006.6  // Marca auxiliar 47
x48              V2006.7  // Marca auxiliar 48
x33              V2007.0  // Marca auxiliar 33
x34              V2007.1  // Marca auxiliar 34
x35              V2007.2  // Marca auxiliar 35
x36              V2007.3  // Marca auxiliar 36
x37              V2007.4  // Marca auxiliar 37
x38              V2007.5  // Marca auxiliar 38
x39              V2007.6  // Marca auxiliar 39
x40              V2007.7  // Marca auxiliar 40
x57              V2008.0  // Marca auxiliar 57
x58              V2008.1  // Marca auxiliar 58
x59              V2008.2  // Marca auxiliar 59
x60              V2008.3  // Marca auxiliar 60
x61              V2008.4  // Marca auxiliar 61
x62              V2008.5  // Marca auxiliar 62
x63              V2008.6  // Marca auxiliar 63
x64              V2008.7  // Marca auxiliar 64
x49              V2009.0  // Marca auxiliar 49
x50              V2009.1  // Marca auxiliar 50
x51              V2009.2  // Marca auxiliar 51
x52              V2009.3  // Marca auxiliar 52
x53              V2009.4  // Marca auxiliar 53
x54              V2009.5  // Marca auxiliar 54
x55              V2009.6  // Marca auxiliar 55
x56              V2009.7  // Marca auxiliar 56
x73              V2010.0  // Marca auxiliar 73
x74              V2010.1  // Marca auxiliar 74
x75              V2010.2  // Marca auxiliar 75
x76              V2010.3  // Marca auxiliar 76
x77              V2010.4  // Marca auxiliar 77
x78              V2010.5  // Marca auxiliar 78
x79              V2010.6  // Marca auxiliar 79
x80              V2010.7  // Marca auxiliar 80
x65              V2011.0  // Marca auxiliar 65
x66              V2011.1  // Marca auxiliar 66
x67              V2011.2  // Marca auxiliar 67
x68              V2011.3  // Marca auxiliar 68
x69              V2011.4  // Marca auxiliar 69
x70              V2011.5  // Marca auxiliar 70
x71              V2011.6  // Marca auxiliar 71
x72              V2011.7  // Marca auxiliar 72
dAux1            VD2012   // Doble palabra de uso comun
ANUsrW00         VW1800   // Version de usuario OP7
ANImgW02         VW1802   // Numero de la imagen
ANImgW04         VW1804   // Numero de la imagen
ANAvsW06         VW1806   // Aviso de servicio 01 a 16
ANAvsW08         VW1808   // Aviso de servicio 07 a 32
ANAvsW10         VW1810   // Aviso de servicio 33 a 48
ANAvsW12         VW1812   // Aviso de servicio 48 a 64
ANAvsW14         VW1814   // Aviso de servicio 65 a 80
ANAvsW16         VW1816   // Aviso de servicio 81 a 96
ANAvsW18         VW1818   // Aviso de servicio 97 a 112
ANAlaW20         VW1820   // Alarmas 01 a 16
ANAlaW22         VW1822   // Alarmas 07 a 32
ANAlaW24         VW1824   // Alarmas 33 a 48
ANAlaW26         VW1826   // Alarmas 48 a 64
ANAlaW28         VW1828   // Alarmas 65 a 80
ANAlaW30         VW1830   // Alarmas 81 a 96
ANAlaW32         VW1832   // Alarmas 97 a 112
ANFalW34         VW1834   // Fallas 01 a 16
ANFalW36         VW1836   // Fallas 07 a 32
ANFalW38         VW1838   // Fallas 33 a 48
ANFalW40         VW1840   // Fallas 48 a 64
ANFalW42         VW1842   // Fallas 65 a 80
ANFalW44         VW1844   // Fallas 81 a 96
ANFalW46         VW1846   // Fallas 97 a 112
ANRecW48         VW1848   // Reconocimientos 01 a 16
ANRecW50         VW1850   // Reconocimientos 07 a 32
ANRecW52         VW1852   // Reconocimientos 33 a 48
ANRecW54         VW1854   // Reconocimientos 48 a 64
ANRecW56         VW1856   // Reconocimientos 65 a 80
ANRecW58         VW1858   // Reconocimientos 81 a 96
ANRecW60         VW1860   // Reconocimientos 97 a 112
TcSisW00         VW1862   // Teclado de sistema Palabra 1
TcSisW02         VW1864   // Teclado de sistema Palabra 2
TcFunW00         VW1866   // Teclado de funciones Palabra 1
TcFunW02         VW1868   // Teclado de funciones Palabra 2
TcFunW04         VW1870   // Teclado de funciones Palabra 3
TcFunW06         VW1872   // Teclado de funciones Palabra 4
ImLedW00         VW1874   // Imagen de los Leds Palabra 1
ImLedW02         VW1876   // Imagen de los Leds Palabra 2
AxSisW00         VW1878   // Auxiliar Teclado de sistema Palabra 1
AxSisW02         VW1880   // Auxiliar Teclado de sistema Palabra 2
AxFunW00         VW1882   // Auxiliar Teclado de funciones Palabra 1
AxFunW02         VW1884   // Auxiliar Teclado de funciones Palabra 2
AxFunW04         VW1886   // Auxiliar Teclado de funciones Palabra 3
AxFunW06         VW1888   // Auxiliar Teclado de funciones Palabra 4
Res1890          VW1890   // Reserva
Res1892          VW1892   // Reserva
fTcSisW00        VW1894   // Flanco Teclado de sistema Palabra 1
fTcSisW02        VW1896   // Flanco Teclado de sistema Palabra 2
fTcFunW00        VW1898   // Flanco Teclado de funciones Palabra 1
fTcFunW02        VW1900   // Flanco Teclado de funciones Palabra 2
fTcFunW04        VW1902   // Flanco Teclado de funciones Palabra 3
fTcFunW06        VW1904   // Flanco Teclado de funciones Palabra 4
wLedRap          VW1996   // Palabra de led rojo permanente
wLedLen          VW1998   // Palabra de led rojo intermitente
wLedPer          VW2000   // Palabra de led verde permanente
wAux1            VW2002   // Palabra auxiliar de uso comun 1
wAux2            VW2004   // Palabra auxiliar de uso comun 2
wAux3            VW2006   // Palabra auxiliar de uso comun 3
wAux4            VW2008   // Palabra auxiliar de uso comun 4
wAux5            VW2010   // Palabra auxiliar de uso comun 5
END_SYMBOL_TABLE

SYMBOL_TABLE Marks Libres
PosicionArmado   VD10     // Valor del Encoder Para Armado
PosicionEncolado VD14     // Valor del Encoder Para Encolado
ReinicioHC0      VD18     // Valor de reinicio del contador rapido HC0
OffSetEncoder    VD22     // Valor de reinicio del contador rapido HC0
PosicionEncoladoOffSet VD26     // Valor del Encoder Para Encolado más Off Set
Cargar_Valor_Encolar M30.0    // Mark Indicadora Cargar valor Posicion Encolar
Cargar_Valor_Armar M30.1    // Mark Indicadora de Posicion Armar
Hay_Caja_Para_Armado M30.2    // Mark Hay Caja para Armado, Habilita Pusher
Area_Armado      M30.3    // Mark Armar
Area_Encolado    M30.4    // Mark Encolar
Parar_Cinta_x_Solapa M30.5    // Mark Parar Cinta Transportadora Por Solapa Trasera Abierta
Subir            M30.6    // Mark Para hacer Subir el brazo
Bajar            M30.7    // Mark Para hacer Bajar el brazo
M_FallaGral      M1.0     // Mark_ParadaGral.Se resetea cuando paso por cero el encoder
Parada_Activada  M31.0    // Mark Stop Presionado
Reconocer_Activado M31.1    // Mark Reconocer Presionado
Mark_Activar_Vacio M31.2    // Mark Activar Vacio
Mark_Act_Solapa_Manual M31.3    // Mark Activar Solapa Trasera (Para Modo Manual)
Ssr_Arriba       M29.0    // Sensor Brazo Arriba
f_Ssr_Pist_Pusher_Atras M29.1    // Flanco Positivo Sensor de Piston del Pusher Atras
END_SYMBOL_TABLE

ORGANIZATION_BLOCK Program_Block:OB1
TITLE=	
// 		***************************************************
// 		********Armadora de cajas Stork 2........******
// 		***************************************************	
// GMG 2005-04-20 
BEGIN
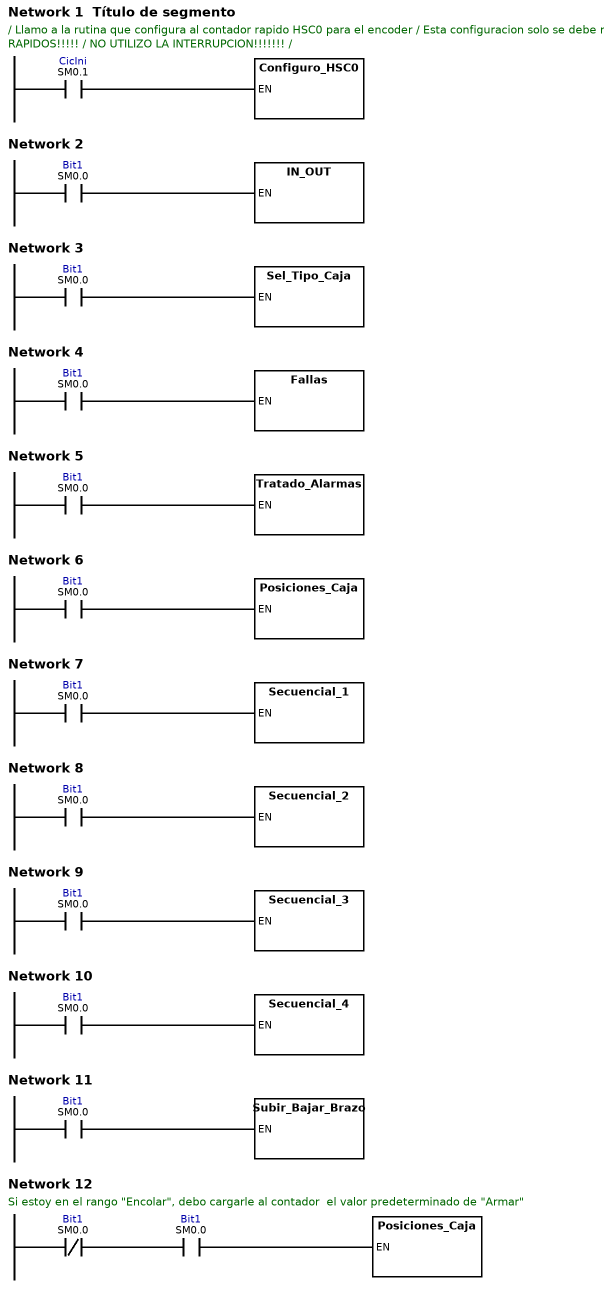
Network 1 // Título de segmento
// 
// Llamo a la rutina que configura al contador rapido HSC0 para el encoder
// Esta configuracion solo se debe realizar en el 1º ciclo!!
// Para mas informacion ver el manual en el capitulo de CONTADORES RAPIDOS!!!!!
// NO UTILIZO LA INTERRUPCION!!!!!!!
// 
LD     CicIni:SM0.1
CALL   Configuro_HSC0:SBR1
Network 2
LD     Bit1:SM0.0
CALL   IN_OUT:SBR2
Network 3
LD     Bit1:SM0.0
CALL   Sel_Tipo_Caja:SBR3
Network 4
LD     Bit1:SM0.0
CALL   Fallas:SBR20
Network 5
LD     Bit1:SM0.0
CALL   Tratado_Alarmas:SBR14
Network 6
LD     Bit1:SM0.0
CALL   Posiciones_Caja:SBR25
Network 7
LD     Bit1:SM0.0
CALL   Secuencial_1:SBR6
Network 8
LD     Bit1:SM0.0
CALL   Secuencial_2:SBR7
Network 9
LD     Bit1:SM0.0
CALL   Secuencial_3:SBR8
Network 10
LD     Bit1:SM0.0
CALL   Secuencial_4:SBR0
Network 11
LD     Bit1:SM0.0
CALL   Subir_Bajar_Brazo:SBR13
Network 12
// Si estoy en el rango "Encolar", debo cargarle al contador  el valor predeterminado de "Armar"
LDN    Bit1:SM0.0
A      Bit1:SM0.0
CALL   Posiciones_Caja:SBR25
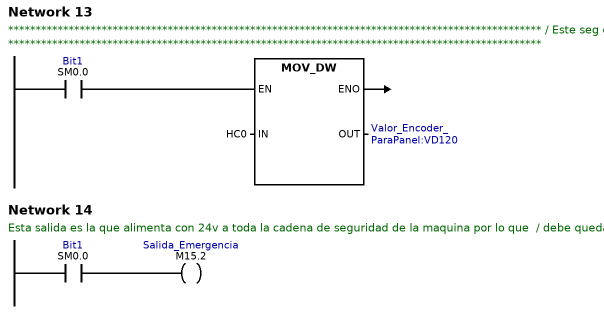
Network 13
// *************************************************************************************************
// Este seg es para poder visualizar en el panel los valores Actuales del Encoder !!!!!!
// *************************************************************************************************
LD     Bit1:SM0.0
MOVD   HC0, Valor_Encoder_ParaPanel:VD120
Network 14
// Esta salida es la que alimenta con 24v a toda la cadena de seguridad de la maquina por lo que 
// debe quedar siempre en forma activa 
LD     Bit1:SM0.0
=      Salida_Emergencia:M15.2
END_ORGANIZATION_BLOCK

SUBROUTINE_BLOCK Secuencial_4:SBR0
TITLE=
BEGIN
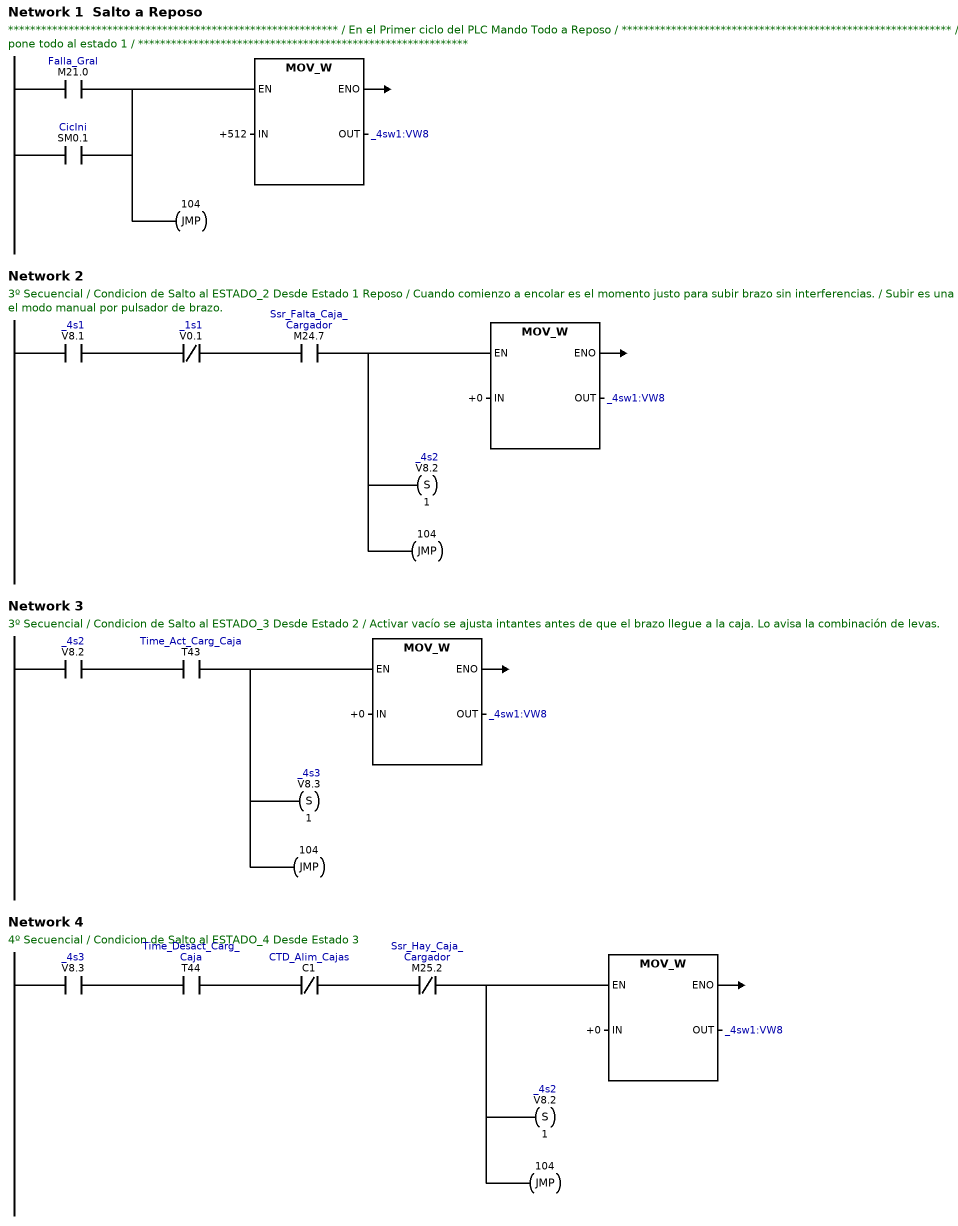
Network 1 // Salto a Reposo
// ************************************************************
// En el Primer ciclo del PLC Mando Todo a Reposo
// ************************************************************
// Si tengo Falla Gral. se pone todo al estado 1
// ************************************************************
LD     Falla_Gral:M21.0
O      CicIni:SM0.1
MOVW   +512, _4sw1:VW8
JMP    104
Network 2
// 3º Secuencial
// Condicion de Salto al ESTADO_2 Desde Estado 1 Reposo
// Cuando comienzo a encolar es el momento justo para subir brazo sin interferencias.
// Subir es una marca que vale solo para el modo manual por pulsador de brazo.
LD     _4s1:V8.1
AN     _1s1:V0.1
A      Ssr_Falta_Caja_Cargador:M24.7
MOVW   +0, _4sw1:VW8
S      _4s2:V8.2, 1
JMP    104
Network 3
// 3º Secuencial
// Condicion de Salto al ESTADO_3 Desde Estado 2
// Activar vacío se ajusta intantes antes de que el brazo llegue a la caja. Lo avisa la combinación de levas.
LD     _4s2:V8.2
A      Time_Act_Carg_Caja:T43
MOVW   +0, _4sw1:VW8
S      _4s3:V8.3, 1
JMP    104
Network 4
// 4º Secuencial
// Condicion de Salto al ESTADO_4 Desde Estado 3
LD     _4s3:V8.3
A      Time_Desact_Carg_Caja:T44
AN     CTD_Alim_Cajas:C1
AN     Ssr_Hay_Caja_Cargador:M25.2
MOVW   +0, _4sw1:VW8
S      _4s2:V8.2, 1
JMP    104
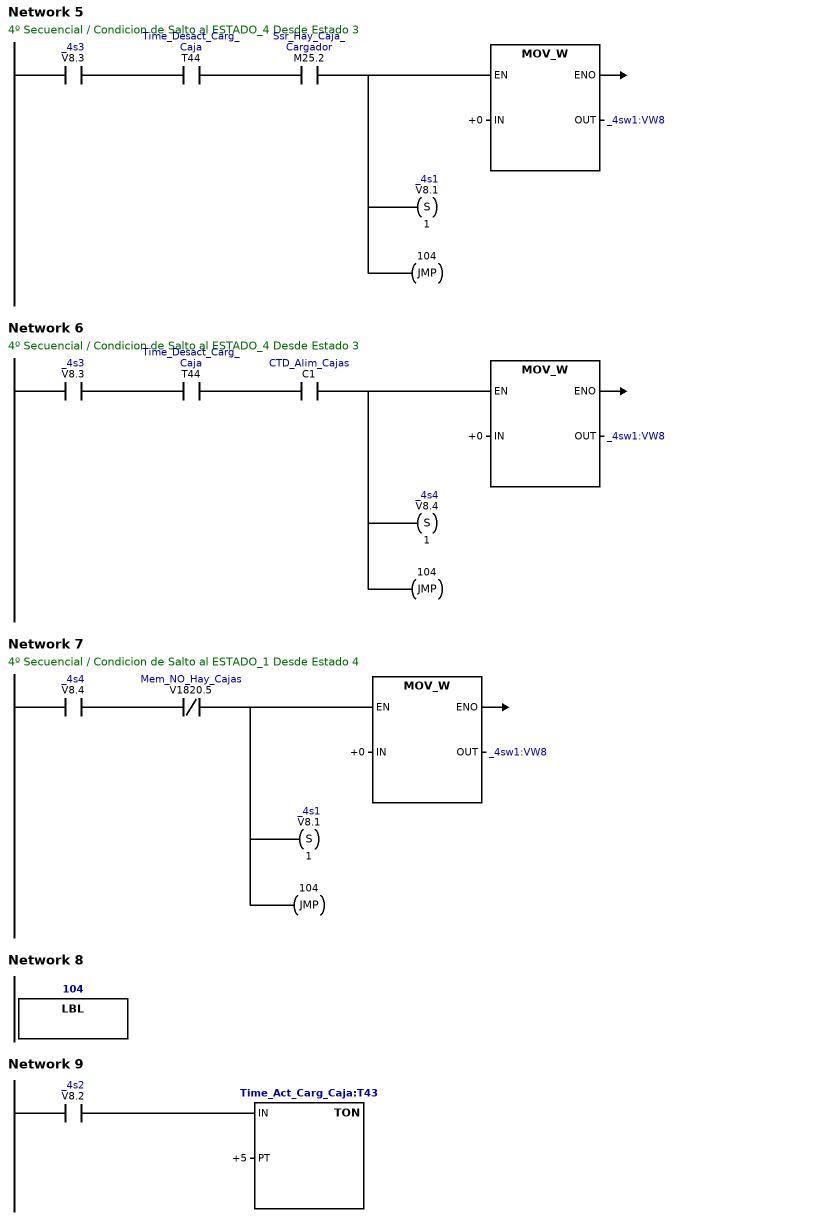
Network 5
// 4º Secuencial
// Condicion de Salto al ESTADO_4 Desde Estado 3
LD     _4s3:V8.3
A      Time_Desact_Carg_Caja:T44
A      Ssr_Hay_Caja_Cargador:M25.2
MOVW   +0, _4sw1:VW8
S      _4s1:V8.1, 1
JMP    104
Network 6
// 4º Secuencial
// Condicion de Salto al ESTADO_4 Desde Estado 3
LD     _4s3:V8.3
A      Time_Desact_Carg_Caja:T44
A      CTD_Alim_Cajas:C1
MOVW   +0, _4sw1:VW8
S      _4s4:V8.4, 1
JMP    104
Network 7
// 4º Secuencial
// Condicion de Salto al ESTADO_1 Desde Estado 4
LD     _4s4:V8.4
AN     Mem_NO_Hay_Cajas:V1820.5
MOVW   +0, _4sw1:VW8
S      _4s1:V8.1, 1
JMP    104
Network 8
LBL    104
Network 9
LD     _4s2:V8.2
TON    Time_Act_Carg_Caja:T43, +5
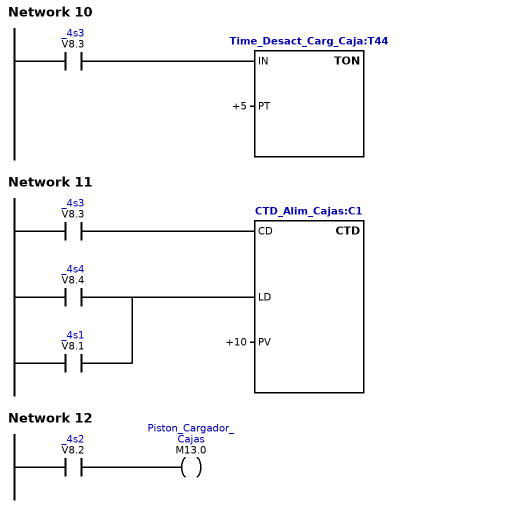
Network 10
LD     _4s3:V8.3
TON    Time_Desact_Carg_Caja:T44, +5
Network 11
LD     _4s3:V8.3
LD     _4s4:V8.4
O      _4s1:V8.1
CTD    CTD_Alim_Cajas:C1, +10
Network 12
LD     _4s2:V8.2
=      Piston_Cargador_Cajas:M13.0
END_SUBROUTINE_BLOCK

SUBROUTINE_BLOCK Configuro_HSC0:SBR1
TITLE=onfiguro El HSC0 en el modo 10 (fases A/B y cero) las palabras especiales son
// 
// SMB37 -> Byte de Control
// SMB36 -> Byte de Estado
// SMD38 -> Nuevo Valor  Actual
// SMD42 -> Nuevo Valor Predeterminado
// 
// Como se utiliza el HSC0 el encoder debe ser conectado en las entradas 
// 
// I0.0 -> Fase A
// I0.1 -> Fase B
// I0.2 -> Puesta a Cero
// 
// Evento de interrupcion 12  -> HSC0  CV=PV no utilizado!!!!
// 
BEGIN
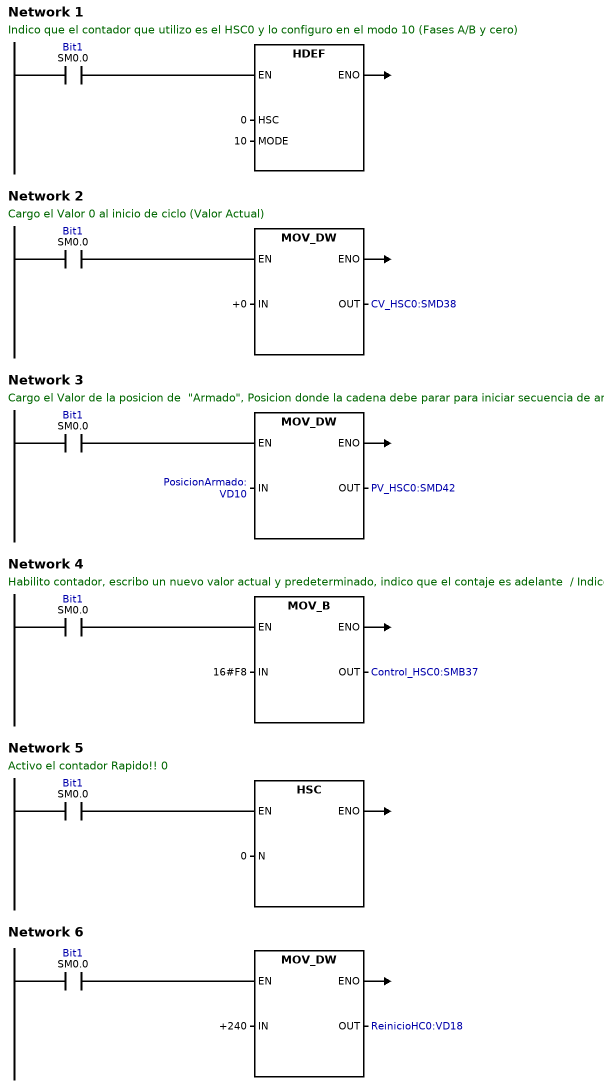
Network 1
// Indico que el contador que utilizo es el HSC0 y lo configuro en el modo 10 (Fases A/B y cero)
LD     Bit1:SM0.0
HDEF   0, 10
Network 2
// Cargo el Valor 0 al inicio de ciclo (Valor Actual)
LD     Bit1:SM0.0
MOVD   +0, CV_HSC0:SMD38
Network 3
// Cargo el Valor de la posicion de  "Armado", Posicion donde la cadena debe parar para iniciar secuencia de armado
LD     Bit1:SM0.0
MOVD   PosicionArmado:VD10, PV_HSC0:SMD42
Network 4
// Habilito contador, escribo un nuevo valor actual y predeterminado, indico que el contaje es adelante 
// Indico actividad alta en las entradas, Cuadruple velocidad
LD     Bit1:SM0.0
MOVB   16#F8, Control_HSC0:SMB37
Network 5
// Activo el contador Rapido!! 0
LD     Bit1:SM0.0
HSC    0
Network 6
LD     Bit1:SM0.0
MOVD   +240, ReinicioHC0:VD18
END_SUBROUTINE_BLOCK

SUBROUTINE_BLOCK IN_OUT:SBR2
TITLE=
BEGIN
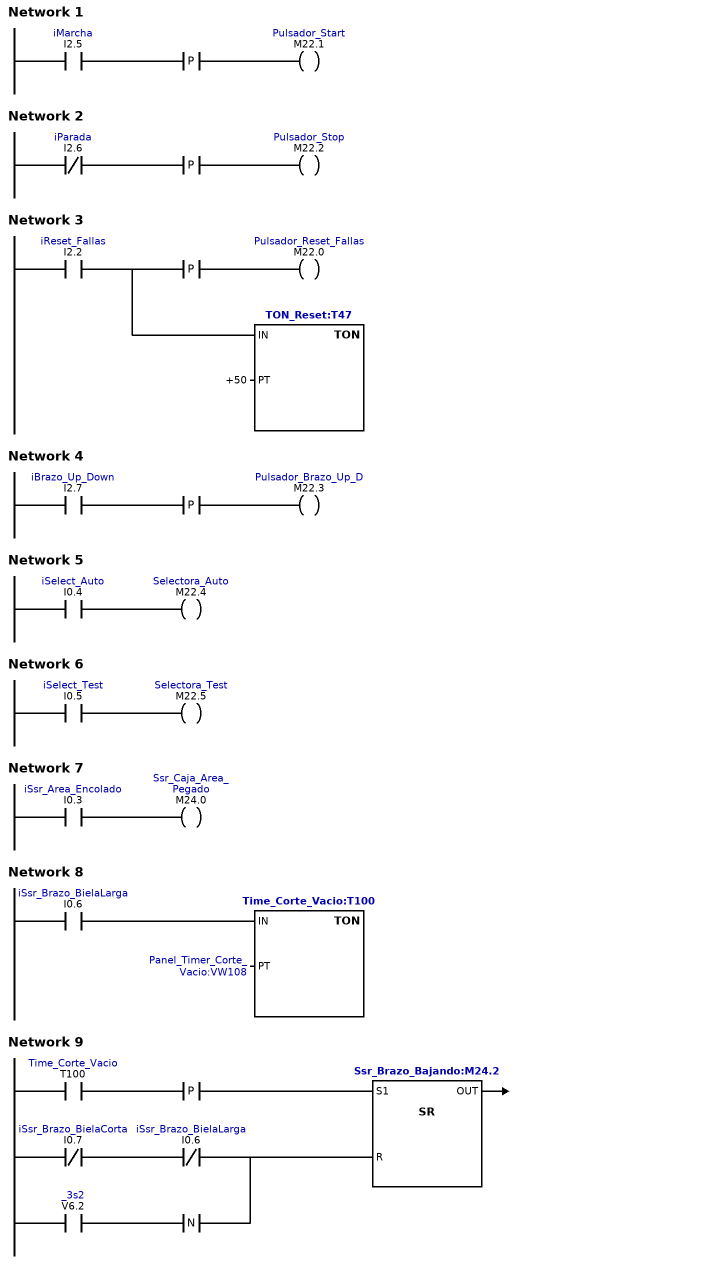
Network 1
LD     iMarcha:I2.5
EU
=      Pulsador_Start:M22.1
Network 2
LDN    iParada:I2.6
EU
=      Pulsador_Stop:M22.2
Network 3
LD     iReset_Fallas:I2.2
LPS
EU
=      Pulsador_Reset_Fallas:M22.0
LPP
TON    TON_Reset:T47, +50
Network 4
LD     iBrazo_Up_Down:I2.7
EU
=      Pulsador_Brazo_Up_D:M22.3
Network 5
LD     iSelect_Auto:I0.4
=      Selectora_Auto:M22.4
Network 6
LD     iSelect_Test:I0.5
=      Selectora_Test:M22.5
Network 7
LD     iSsr_Area_Encolado:I0.3
=      Ssr_Caja_Area_Pegado:M24.0
Network 8
LD     iSsr_Brazo_BielaLarga:I0.6
TON    Time_Corte_Vacio:T100, Panel_Timer_Corte_Vacio:VW108
Network 9
LD     Time_Corte_Vacio:T100
EU
LDN    iSsr_Brazo_BielaCorta:I0.7
AN     iSsr_Brazo_BielaLarga:I0.6
LD     _3s2:V6.2
ED
OLD
NOT
A      Ssr_Brazo_Bajando:M24.2
OLD
=      Ssr_Brazo_Bajando:M24.2
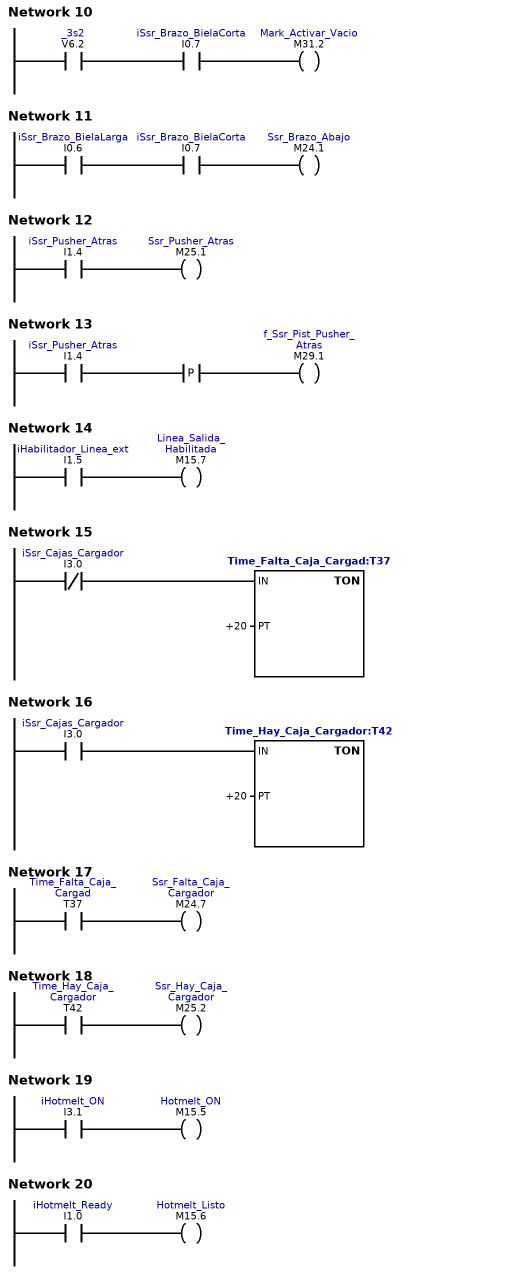
Network 10
LD     _3s2:V6.2
A      iSsr_Brazo_BielaCorta:I0.7
=      Mark_Activar_Vacio:M31.2
Network 11
LD     iSsr_Brazo_BielaLarga:I0.6
A      iSsr_Brazo_BielaCorta:I0.7
=      Ssr_Brazo_Abajo:M24.1
Network 12
LD     iSsr_Pusher_Atras:I1.4
=      Ssr_Pusher_Atras:M25.1
Network 13
LD     iSsr_Pusher_Atras:I1.4
EU
=      f_Ssr_Pist_Pusher_Atras:M29.1
Network 14
LD     iHabilitador_Linea_ext:I1.5
=      Linea_Salida_Habilitada:M15.7
Network 15
LDN    iSsr_Cajas_Cargador:I3.0
TON    Time_Falta_Caja_Cargad:T37, +20
Network 16
LD     iSsr_Cajas_Cargador:I3.0
TON    Time_Hay_Caja_Cargador:T42, +20
Network 17
LD     Time_Falta_Caja_Cargad:T37
=      Ssr_Falta_Caja_Cargador:M24.7
Network 18
LD     Time_Hay_Caja_Cargador:T42
=      Ssr_Hay_Caja_Cargador:M25.2
Network 19
LD     iHotmelt_ON:I3.1
=      Hotmelt_ON:M15.5
Network 20
LD     iHotmelt_Ready:I1.0
=      Hotmelt_Listo:M15.6
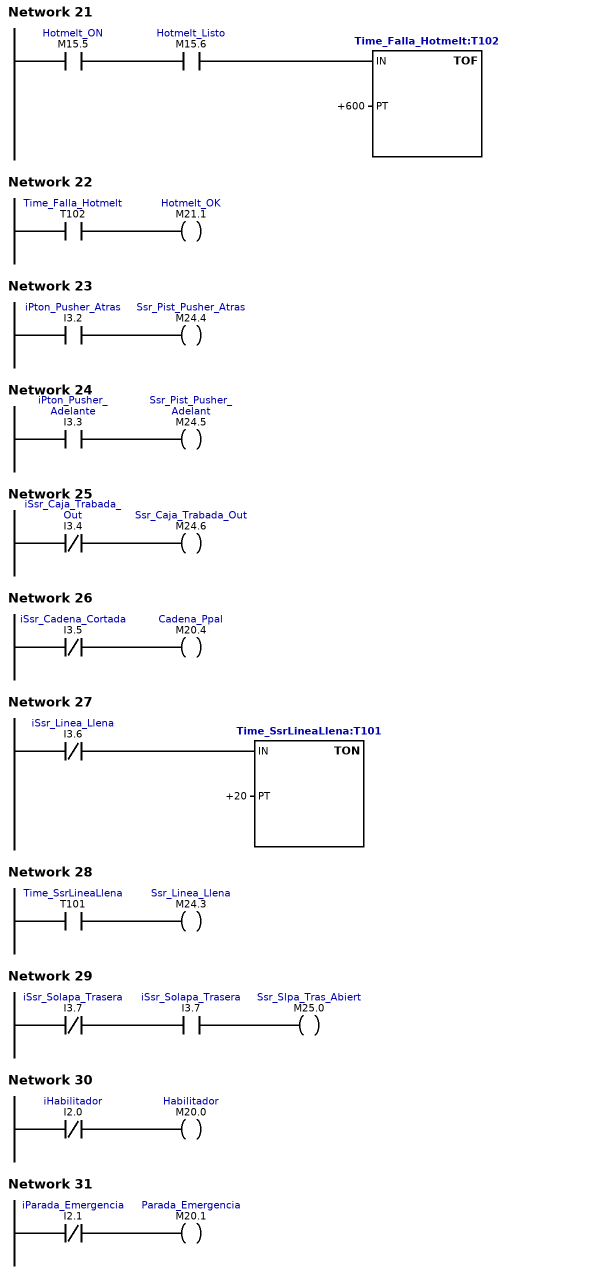
Network 21
LD     Hotmelt_ON:M15.5
A      Hotmelt_Listo:M15.6
TOF    Time_Falla_Hotmelt:T102, +600
Network 22
LD     Time_Falla_Hotmelt:T102
=      Hotmelt_OK:M21.1
Network 23
LD     iPton_Pusher_Atras:I3.2
=      Ssr_Pist_Pusher_Atras:M24.4
Network 24
LD     iPton_Pusher_Adelante:I3.3
=      Ssr_Pist_Pusher_Adelant:M24.5
Network 25
LDN    iSsr_Caja_Trabada_Out:I3.4
=      Ssr_Caja_Trabada_Out:M24.6
Network 26
LDN    iSsr_Cadena_Cortada:I3.5
=      Cadena_Ppal:M20.4
Network 27
LDN    iSsr_Linea_Llena:I3.6
TON    Time_SsrLineaLlena:T101, +20
Network 28
LD     Time_SsrLineaLlena:T101
=      Ssr_Linea_Llena:M24.3
Network 29
LDN    iSsr_Solapa_Trasera:I3.7
A      iSsr_Solapa_Trasera:I3.7
=      Ssr_Slpa_Tras_Abiert:M25.0
Network 30
LDN    iHabilitador:I2.0
=      Habilitador:M20.0
Network 31
LDN    iParada_Emergencia:I2.1
=      Parada_Emergencia:M20.1
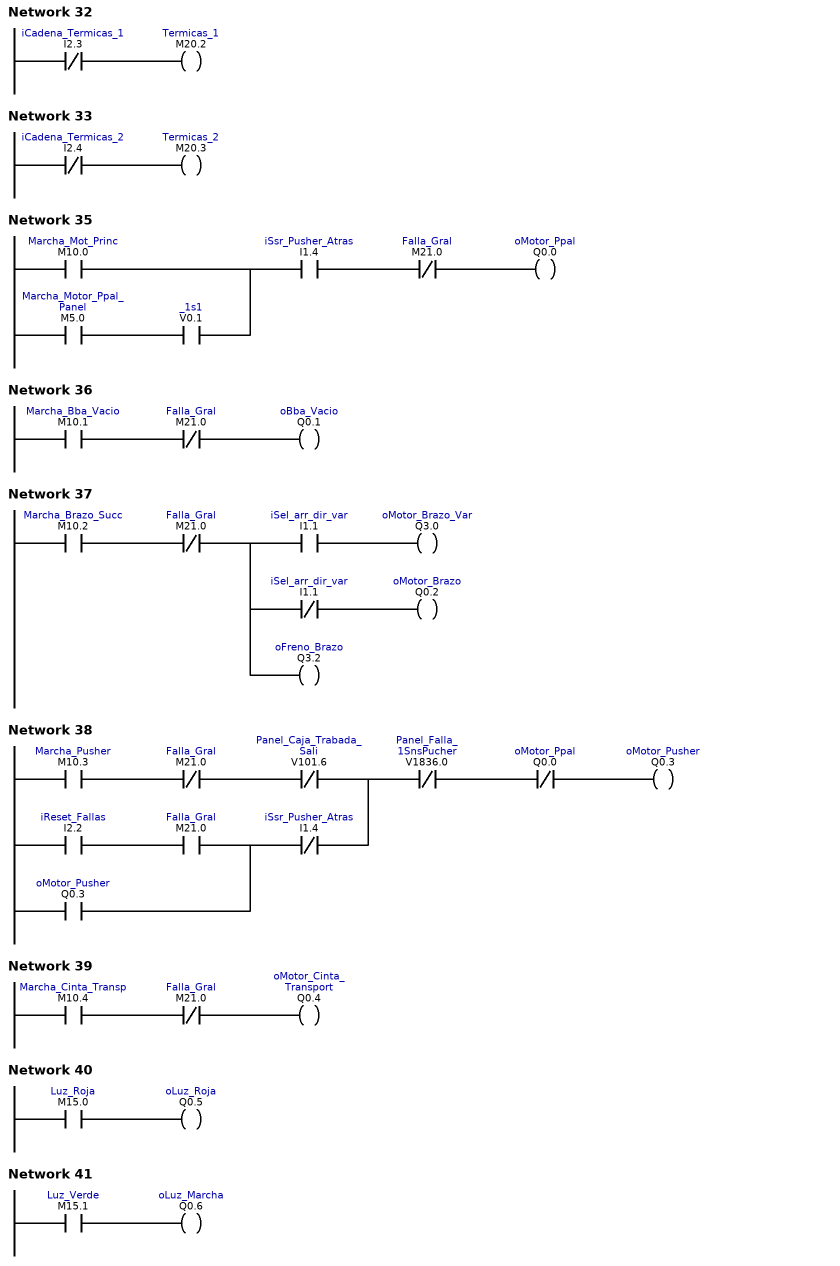
Network 32
LDN    iCadena_Termicas_1:I2.3
=      Termicas_1:M20.2
Network 33
LDN    iCadena_Termicas_2:I2.4
=      Termicas_2:M20.3
Network 35
LD     Marcha_Mot_Princ:M10.0
LD     Marcha_Motor_Ppal_Panel:M5.0
A      _1s1:V0.1
OLD
A      iSsr_Pusher_Atras:I1.4
AN     Falla_Gral:M21.0
=      oMotor_Ppal:Q0.0
Network 36
LD     Marcha_Bba_Vacio:M10.1
AN     Falla_Gral:M21.0
=      oBba_Vacio:Q0.1
Network 37
LD     Marcha_Brazo_Succ:M10.2
AN     Falla_Gral:M21.0
LPS
A      iSel_arr_dir_var:I1.1
=      oMotor_Brazo_Var:Q3.0
LRD
AN     iSel_arr_dir_var:I1.1
=      oMotor_Brazo:Q0.2
LPP
=      oFreno_Brazo:Q3.2
Network 38
LD     Marcha_Pusher:M10.3
AN     Falla_Gral:M21.0
AN     Panel_Caja_Trabada_Sali:V101.6
LD     iReset_Fallas:I2.2
A      Falla_Gral:M21.0
O      oMotor_Pusher:Q0.3
AN     iSsr_Pusher_Atras:I1.4
OLD
AN     Panel_Falla_1SnsPucher:V1836.0
AN     oMotor_Ppal:Q0.0
=      oMotor_Pusher:Q0.3
Network 39
LD     Marcha_Cinta_Transp:M10.4
AN     Falla_Gral:M21.0
=      oMotor_Cinta_Transport:Q0.4
Network 40
LD     Luz_Roja:M15.0
=      oLuz_Roja:Q0.5
Network 41
LD     Luz_Verde:M15.1
=      oLuz_Marcha:Q0.6
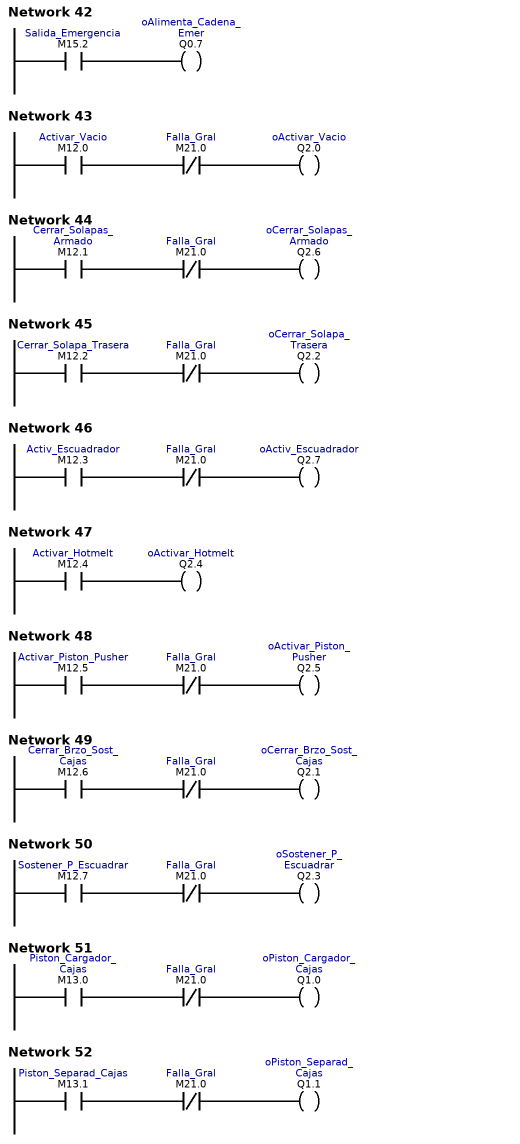
Network 42
LD     Salida_Emergencia:M15.2
=      oAlimenta_Cadena_Emer:Q0.7
Network 43
LD     Activar_Vacio:M12.0
AN     Falla_Gral:M21.0
=      oActivar_Vacio:Q2.0
Network 44
LD     Cerrar_Solapas_Armado:M12.1
AN     Falla_Gral:M21.0
=      oCerrar_Solapas_Armado:Q2.6
Network 45
LD     Cerrar_Solapa_Trasera:M12.2
AN     Falla_Gral:M21.0
=      oCerrar_Solapa_Trasera:Q2.2
Network 46
LD     Activ_Escuadrador:M12.3
AN     Falla_Gral:M21.0
=      oActiv_Escuadrador:Q2.7
Network 47
LD     Activar_Hotmelt:M12.4
=      oActivar_Hotmelt:Q2.4
Network 48
LD     Activar_Piston_Pusher:M12.5
AN     Falla_Gral:M21.0
=      oActivar_Piston_Pusher:Q2.5
Network 49
LD     Cerrar_Brzo_Sost_Cajas:M12.6
AN     Falla_Gral:M21.0
=      oCerrar_Brzo_Sost_Cajas:Q2.1
Network 50
LD     Sostener_P_Escuadrar:M12.7
AN     Falla_Gral:M21.0
=      oSostener_P_Escuadrar:Q2.3
Network 51
LD     Piston_Cargador_Cajas:M13.0
AN     Falla_Gral:M21.0
=      oPiston_Cargador_Cajas:Q1.0
Network 52
LD     Piston_Separad_Cajas:M13.1
AN     Falla_Gral:M21.0
=      oPiston_Separad_Cajas:Q1.1
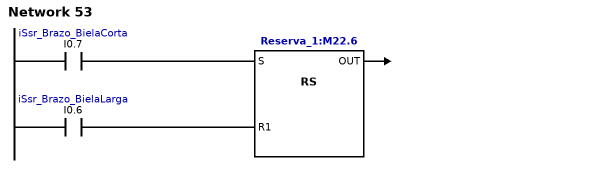
Network 53
LD     iSsr_Brazo_BielaCorta:I0.7
LD     iSsr_Brazo_BielaLarga:I0.6
NOT
LPS
A      Reserva_1:M22.6
=      Reserva_1:M22.6
LPP
ALD
O      Reserva_1:M22.6
=      Reserva_1:M22.6
END_SUBROUTINE_BLOCK

SUBROUTINE_BLOCK Sel_Tipo_Caja:SBR3
TITLE=
BEGIN
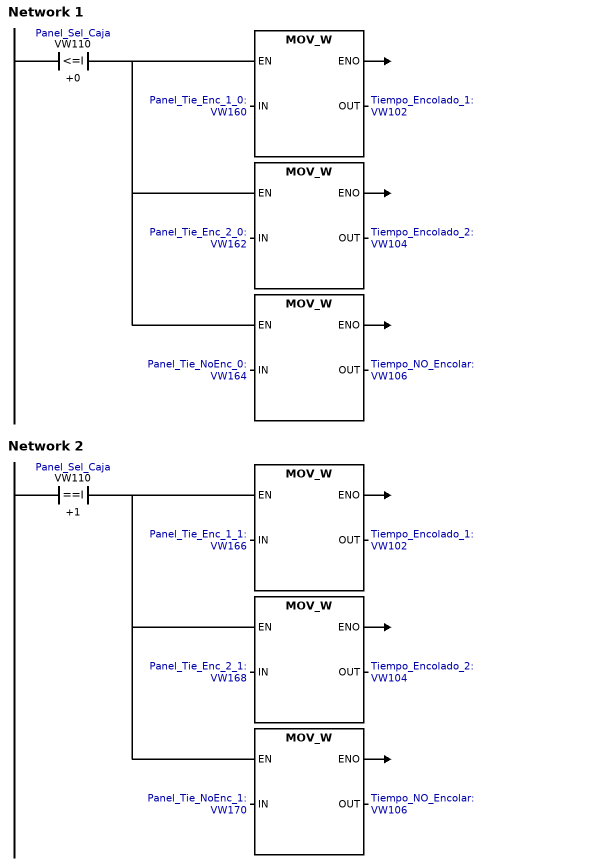
Network 1
LDW<=  Panel_Sel_Caja:VW110, +0
MOVW   Panel_Tie_Enc_1_0:VW160, Tiempo_Encolado_1:VW102
MOVW   Panel_Tie_Enc_2_0:VW162, Tiempo_Encolado_2:VW104
MOVW   Panel_Tie_NoEnc_0:VW164, Tiempo_NO_Encolar:VW106
Network 2
LDW=   Panel_Sel_Caja:VW110, +1
MOVW   Panel_Tie_Enc_1_1:VW166, Tiempo_Encolado_1:VW102
MOVW   Panel_Tie_Enc_2_1:VW168, Tiempo_Encolado_2:VW104
MOVW   Panel_Tie_NoEnc_1:VW170, Tiempo_NO_Encolar:VW106
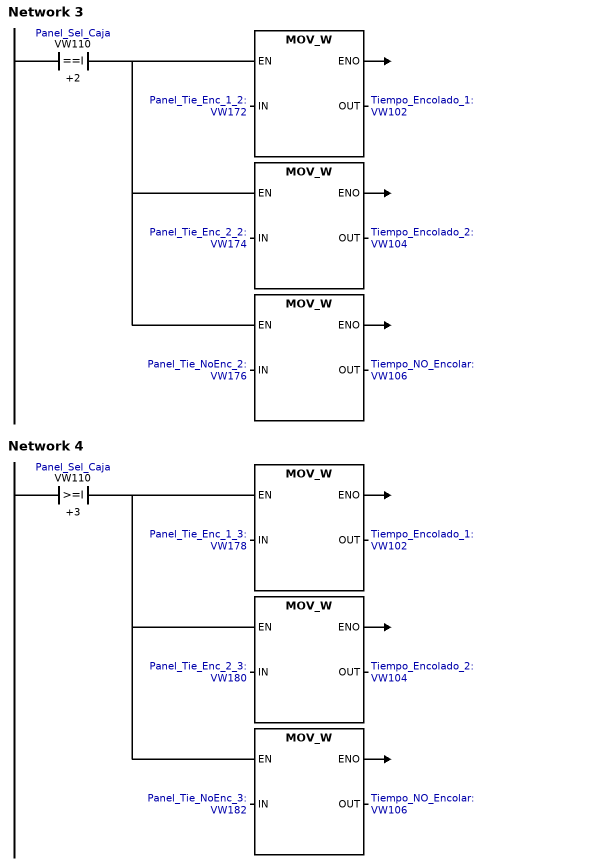
Network 3
LDW=   Panel_Sel_Caja:VW110, +2
MOVW   Panel_Tie_Enc_1_2:VW172, Tiempo_Encolado_1:VW102
MOVW   Panel_Tie_Enc_2_2:VW174, Tiempo_Encolado_2:VW104
MOVW   Panel_Tie_NoEnc_2:VW176, Tiempo_NO_Encolar:VW106
Network 4
LDW>=  Panel_Sel_Caja:VW110, +3
MOVW   Panel_Tie_Enc_1_3:VW178, Tiempo_Encolado_1:VW102
MOVW   Panel_Tie_Enc_2_3:VW180, Tiempo_Encolado_2:VW104
MOVW   Panel_Tie_NoEnc_3:VW182, Tiempo_NO_Encolar:VW106
END_SUBROUTINE_BLOCK

SUBROUTINE_BLOCK Secuencial_1:SBR6
TITLE=
BEGIN
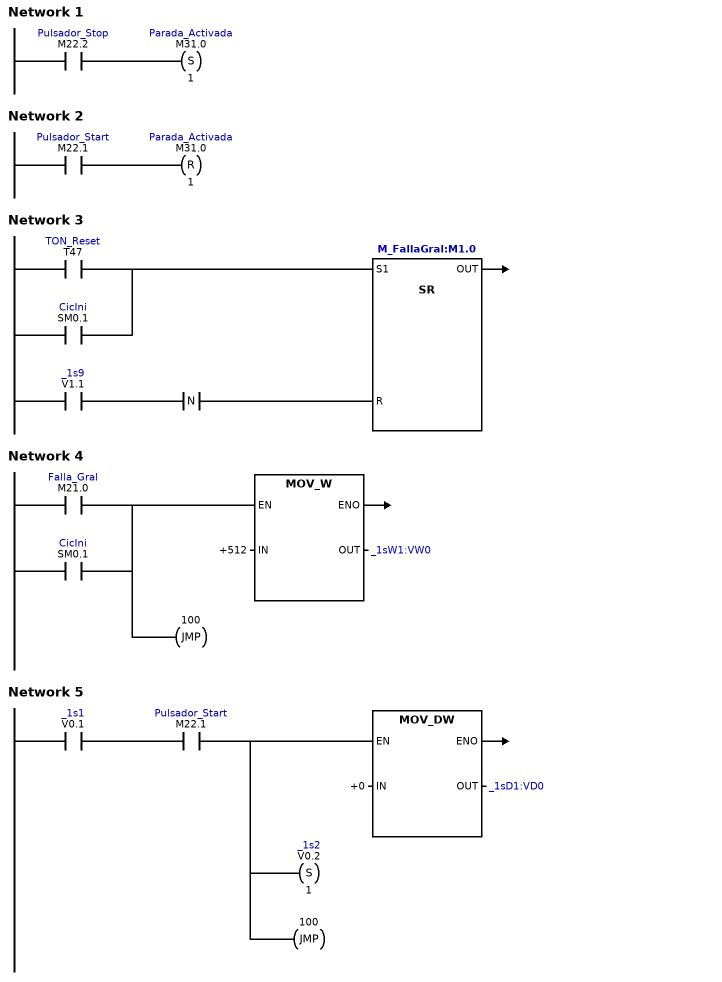
Network 1
LD     Pulsador_Stop:M22.2
S      Parada_Activada:M31.0, 1
Network 2
LD     Pulsador_Start:M22.1
R      Parada_Activada:M31.0, 1
Network 3
LD     TON_Reset:T47
O      CicIni:SM0.1
LD     _1s9:V1.1
ED
NOT
A      M_FallaGral:M1.0
OLD
=      M_FallaGral:M1.0
Network 4
LD     Falla_Gral:M21.0
O      CicIni:SM0.1
MOVW   +512, _1sW1:VW0
JMP    100
Network 5
LD     _1s1:V0.1
A      Pulsador_Start:M22.1
MOVD   +0, _1sD1:VD0
S      _1s2:V0.2, 1
JMP    100
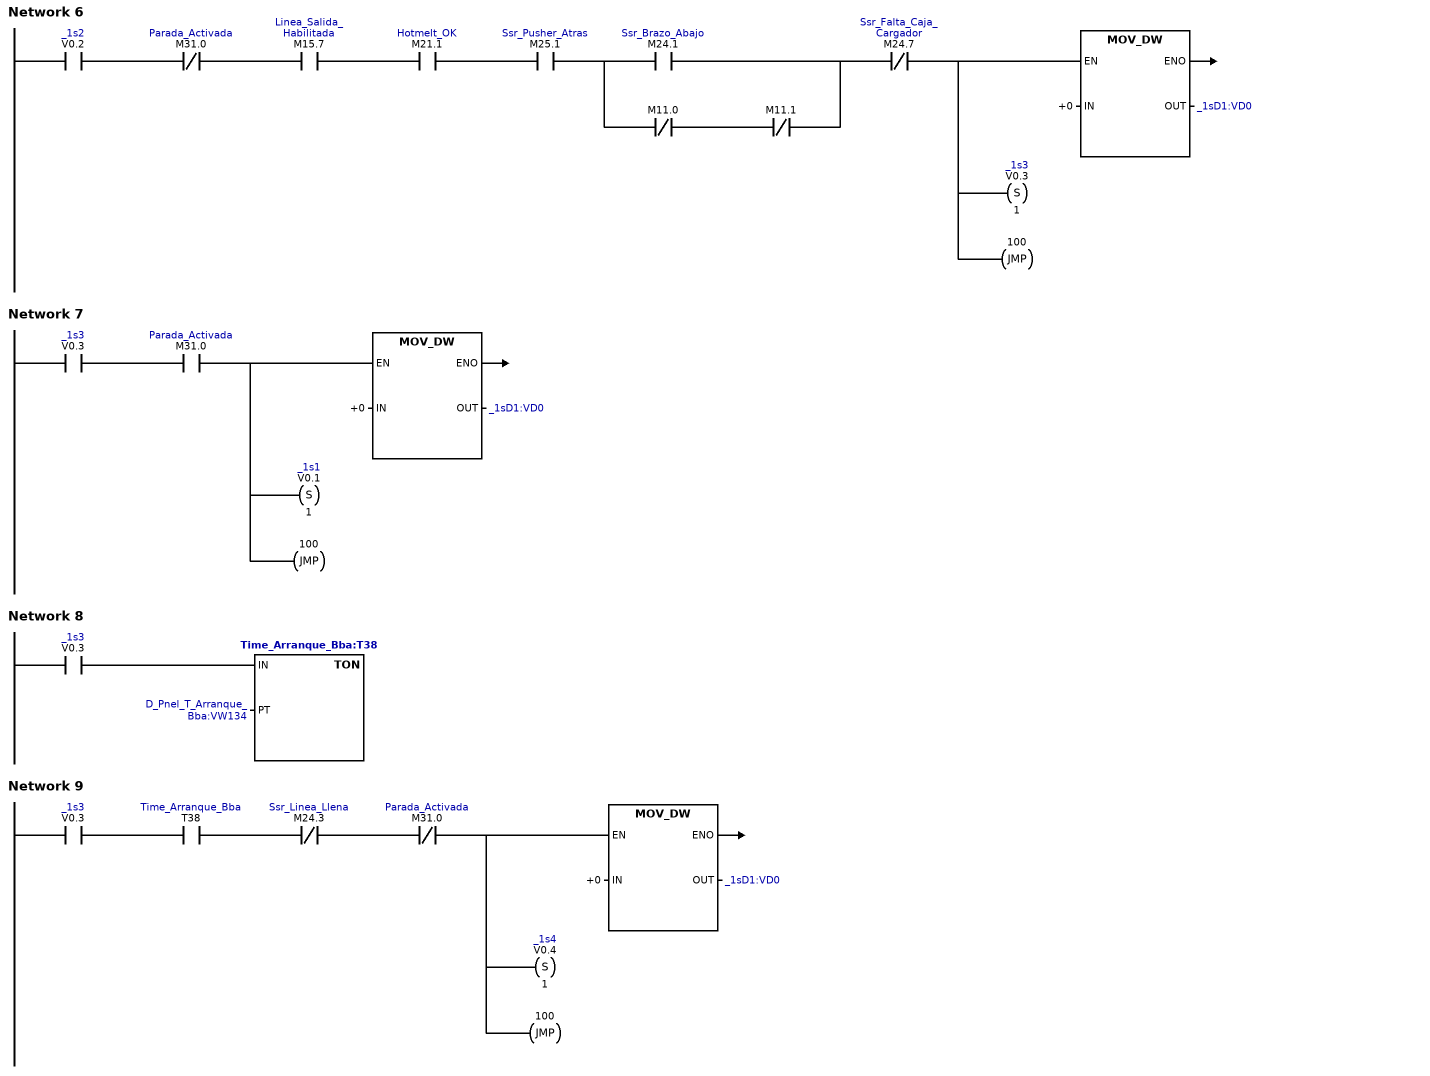
Network 6
LD     _1s2:V0.2
AN     Parada_Activada:M31.0
A      Linea_Salida_Habilitada:M15.7
A      Hotmelt_OK:M21.1
A      Ssr_Pusher_Atras:M25.1
LD     Ssr_Brazo_Abajo:M24.1
LDN    M11.0
AN     M11.1
OLD
ALD
AN     Ssr_Falta_Caja_Cargador:M24.7
MOVD   +0, _1sD1:VD0
S      _1s3:V0.3, 1
JMP    100
Network 7
LD     _1s3:V0.3
A      Parada_Activada:M31.0
MOVD   +0, _1sD1:VD0
S      _1s1:V0.1, 1
JMP    100
Network 8
LD     _1s3:V0.3
TON    Time_Arranque_Bba:T38, D_Pnel_T_Arranque_Bba:VW134
Network 9
LD     _1s3:V0.3
A      Time_Arranque_Bba:T38
AN     Ssr_Linea_Llena:M24.3
AN     Parada_Activada:M31.0
MOVD   +0, _1sD1:VD0
S      _1s4:V0.4, 1
JMP    100
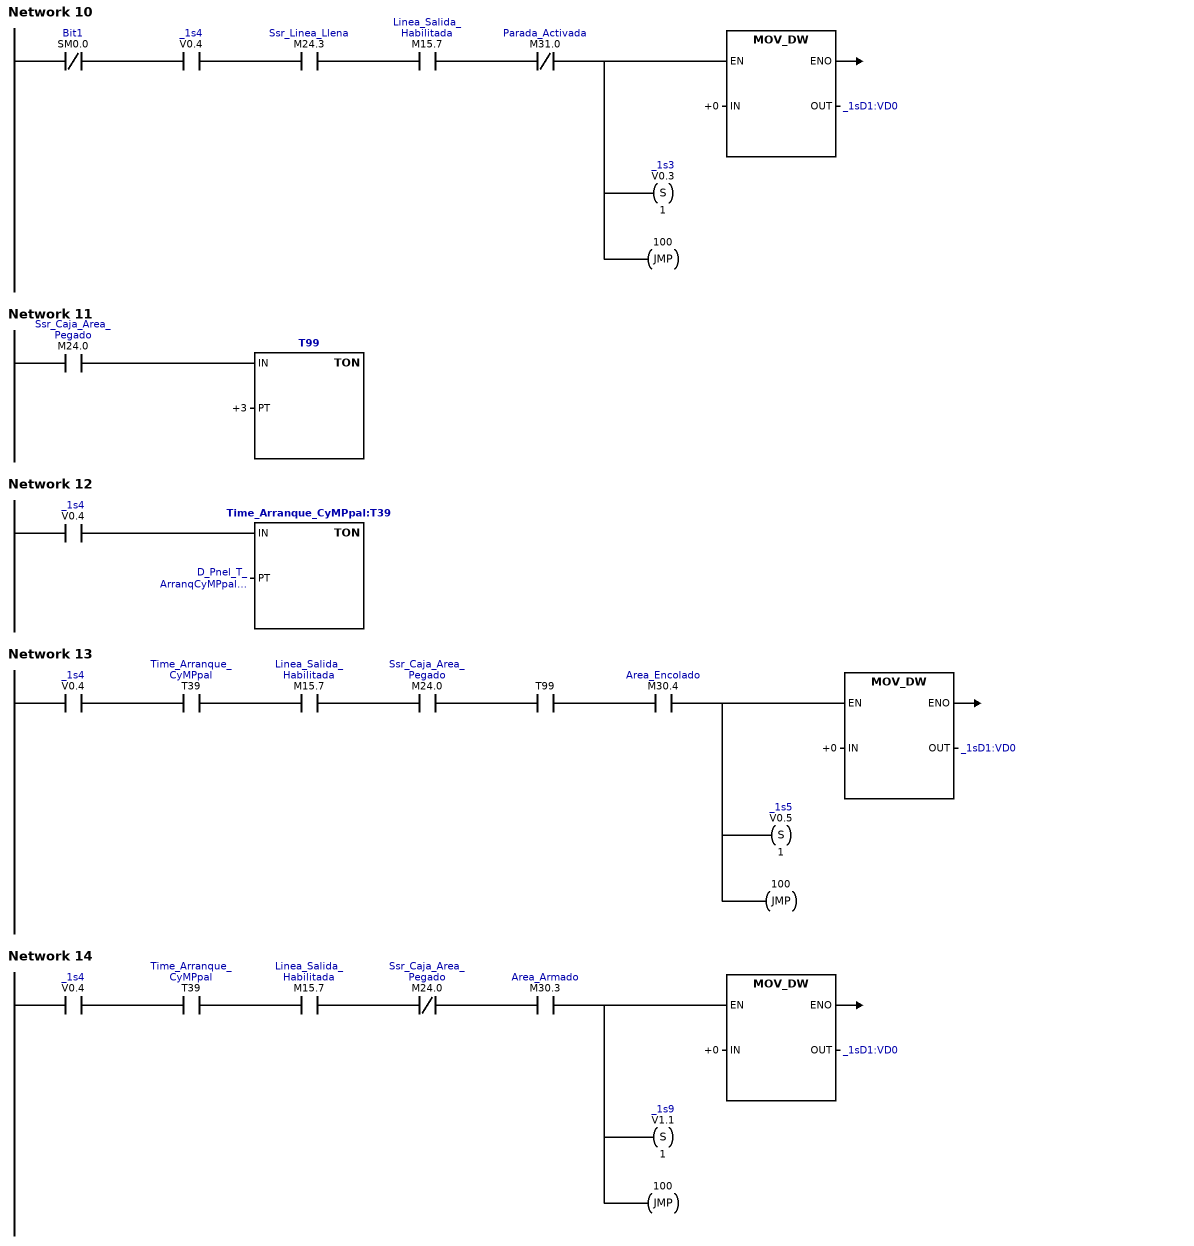
Network 10
LDN    Bit1:SM0.0
A      _1s4:V0.4
A      Ssr_Linea_Llena:M24.3
A      Linea_Salida_Habilitada:M15.7
AN     Parada_Activada:M31.0
MOVD   +0, _1sD1:VD0
S      _1s3:V0.3, 1
JMP    100
Network 11
LD     Ssr_Caja_Area_Pegado:M24.0
TON    T99, +3
Network 12
LD     _1s4:V0.4
TON    Time_Arranque_CyMPpal:T39, D_Pnel_T_ArranqCyMPpal:VW136
Network 13
LD     _1s4:V0.4
A      Time_Arranque_CyMPpal:T39
A      Linea_Salida_Habilitada:M15.7
A      Ssr_Caja_Area_Pegado:M24.0
A      T99
A      Area_Encolado:M30.4
MOVD   +0, _1sD1:VD0
S      _1s5:V0.5, 1
JMP    100
Network 14
LD     _1s4:V0.4
A      Time_Arranque_CyMPpal:T39
A      Linea_Salida_Habilitada:M15.7
AN     Ssr_Caja_Area_Pegado:M24.0
A      Area_Armado:M30.3
MOVD   +0, _1sD1:VD0
S      _1s9:V1.1, 1
JMP    100
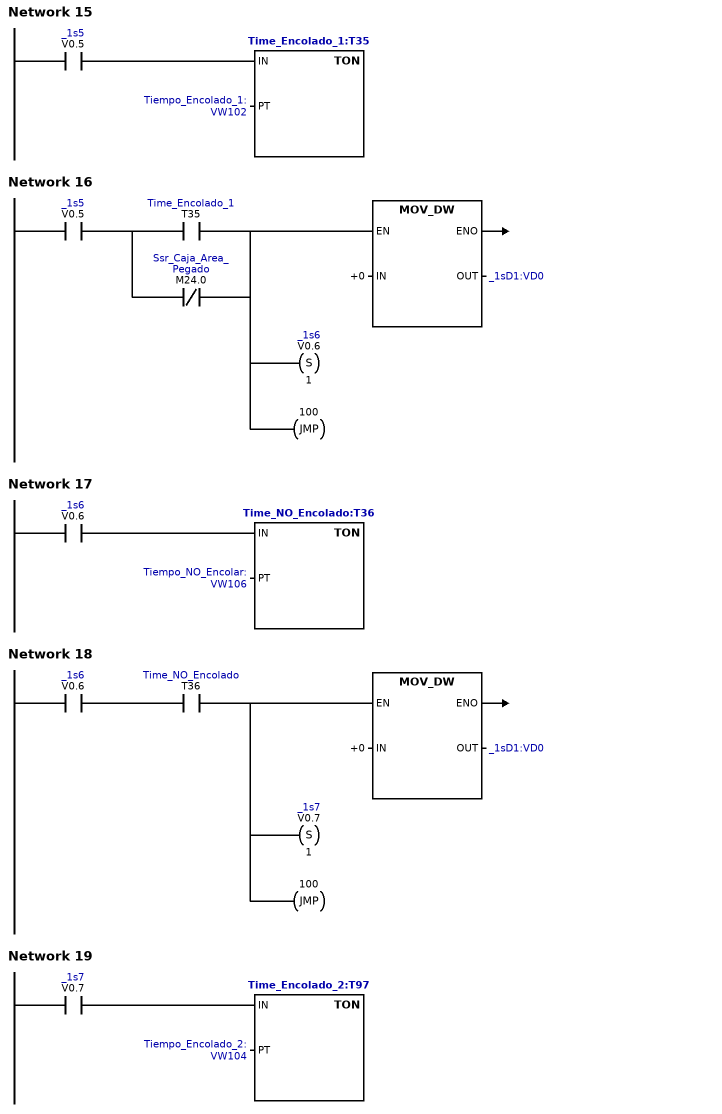
Network 15
LD     _1s5:V0.5
TON    Time_Encolado_1:T35, Tiempo_Encolado_1:VW102
Network 16
LD     _1s5:V0.5
LD     Time_Encolado_1:T35
ON     Ssr_Caja_Area_Pegado:M24.0
ALD
MOVD   +0, _1sD1:VD0
S      _1s6:V0.6, 1
JMP    100
Network 17
LD     _1s6:V0.6
TON    Time_NO_Encolado:T36, Tiempo_NO_Encolar:VW106
Network 18
LD     _1s6:V0.6
A      Time_NO_Encolado:T36
MOVD   +0, _1sD1:VD0
S      _1s7:V0.7, 1
JMP    100
Network 19
LD     _1s7:V0.7
TON    Time_Encolado_2:T97, Tiempo_Encolado_2:VW104
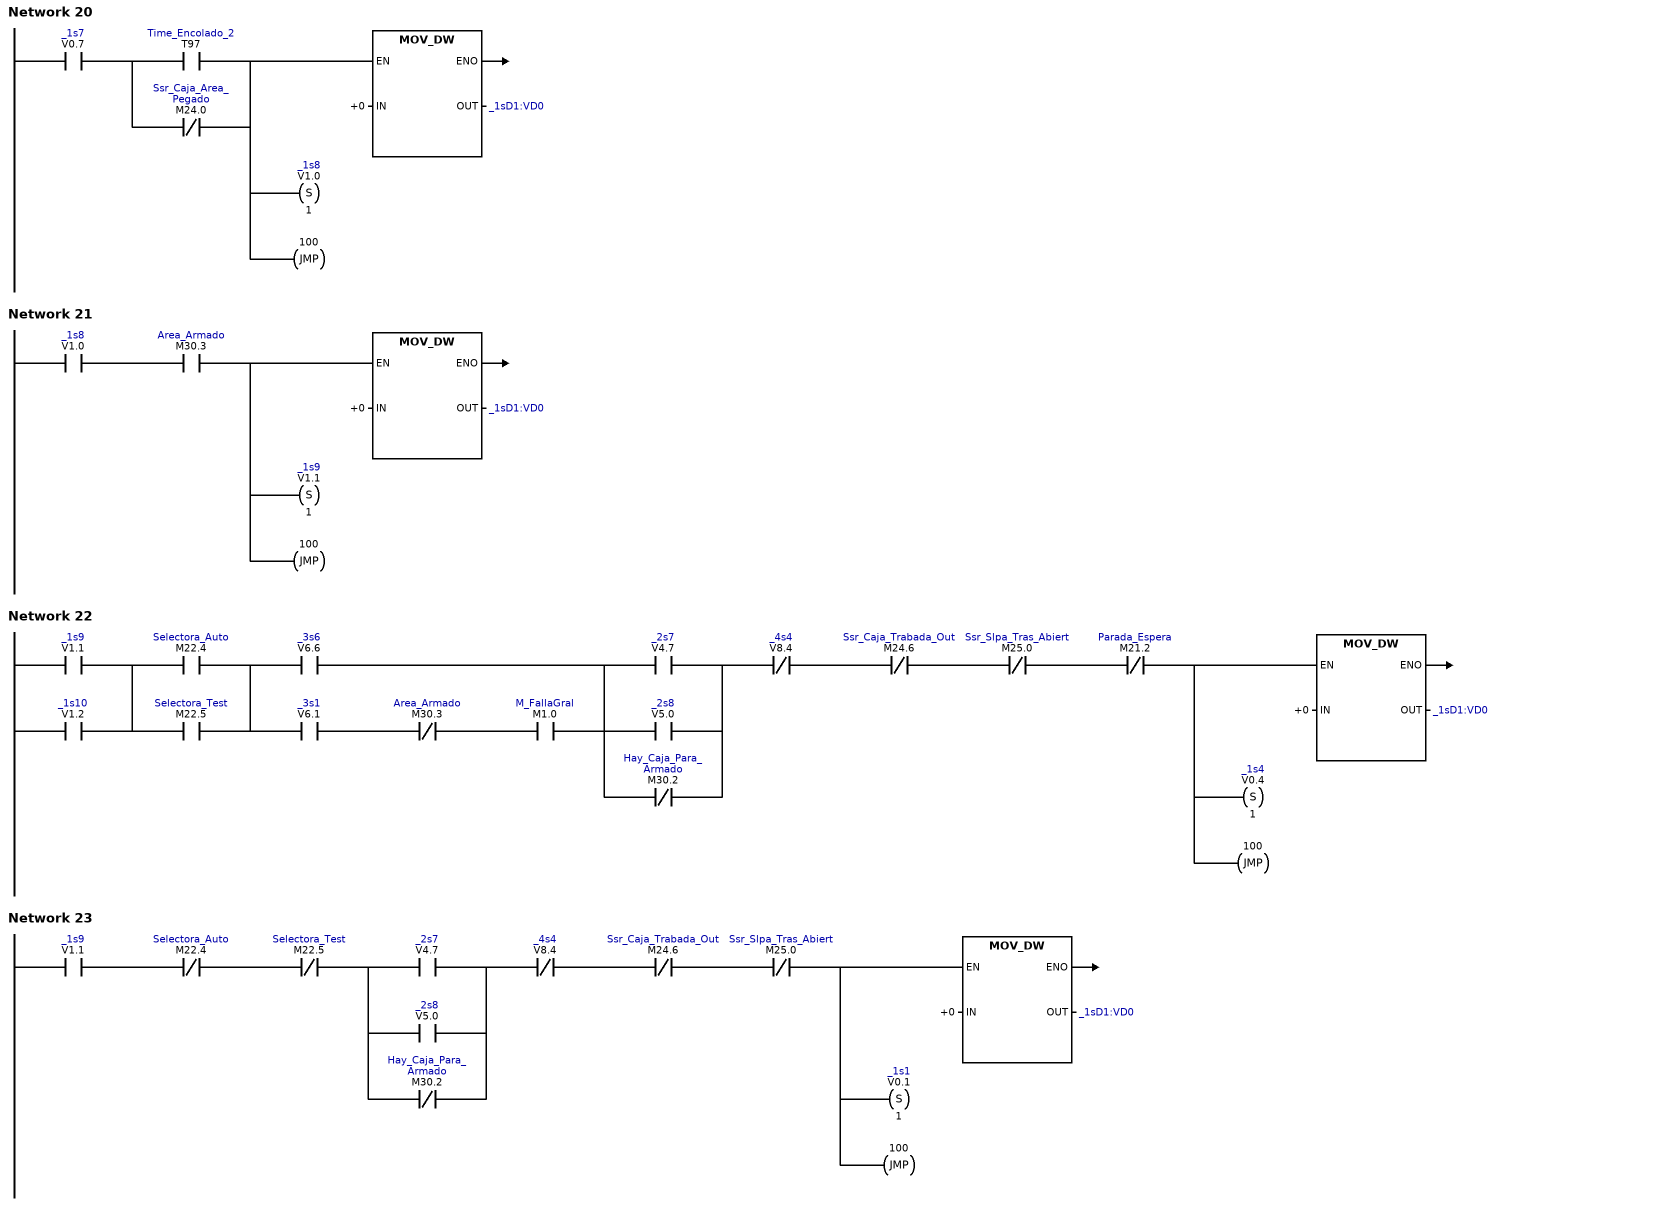
Network 20
LD     _1s7:V0.7
LD     Time_Encolado_2:T97
ON     Ssr_Caja_Area_Pegado:M24.0
ALD
MOVD   +0, _1sD1:VD0
S      _1s8:V1.0, 1
JMP    100
Network 21
LD     _1s8:V1.0
A      Area_Armado:M30.3
MOVD   +0, _1sD1:VD0
S      _1s9:V1.1, 1
JMP    100
Network 22
LD     _1s9:V1.1
O      _1s10:V1.2
LD     Selectora_Auto:M22.4
O      Selectora_Test:M22.5
ALD
LD     _3s6:V6.6
LD     _3s1:V6.1
AN     Area_Armado:M30.3
A      M_FallaGral:M1.0
OLD
ALD
LD     _2s7:V4.7
O      _2s8:V5.0
ON     Hay_Caja_Para_Armado:M30.2
ALD
AN     _4s4:V8.4
AN     Ssr_Caja_Trabada_Out:M24.6
AN     Ssr_Slpa_Tras_Abiert:M25.0
AN     Parada_Espera:M21.2
MOVD   +0, _1sD1:VD0
S      _1s4:V0.4, 1
JMP    100
Network 23
LD     _1s9:V1.1
AN     Selectora_Auto:M22.4
AN     Selectora_Test:M22.5
LD     _2s7:V4.7
O      _2s8:V5.0
ON     Hay_Caja_Para_Armado:M30.2
ALD
AN     _4s4:V8.4
AN     Ssr_Caja_Trabada_Out:M24.6
AN     Ssr_Slpa_Tras_Abiert:M25.0
MOVD   +0, _1sD1:VD0
S      _1s1:V0.1, 1
JMP    100
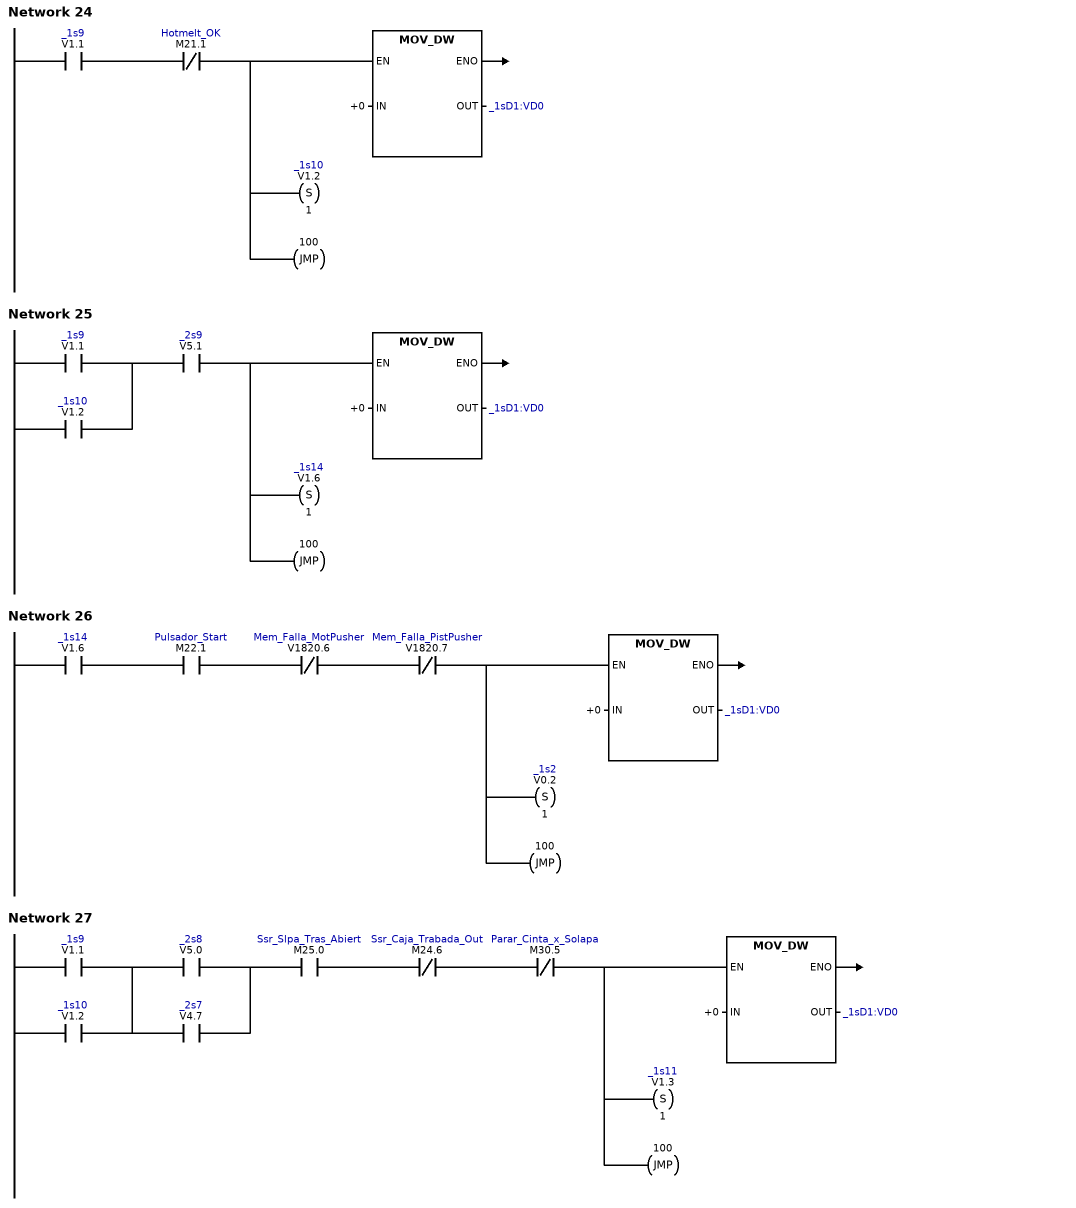
Network 24
LD     _1s9:V1.1
AN     Hotmelt_OK:M21.1
MOVD   +0, _1sD1:VD0
S      _1s10:V1.2, 1
JMP    100
Network 25
LD     _1s9:V1.1
O      _1s10:V1.2
A      _2s9:V5.1
MOVD   +0, _1sD1:VD0
S      _1s14:V1.6, 1
JMP    100
Network 26
LD     _1s14:V1.6
A      Pulsador_Start:M22.1
AN     Mem_Falla_MotPusher:V1820.6
AN     Mem_Falla_PistPusher:V1820.7
MOVD   +0, _1sD1:VD0
S      _1s2:V0.2, 1
JMP    100
Network 27
LD     _1s9:V1.1
O      _1s10:V1.2
LD     _2s8:V5.0
O      _2s7:V4.7
ALD
A      Ssr_Slpa_Tras_Abiert:M25.0
AN     Ssr_Caja_Trabada_Out:M24.6
AN     Parar_Cinta_x_Solapa:M30.5
MOVD   +0, _1sD1:VD0
S      _1s11:V1.3, 1
JMP    100
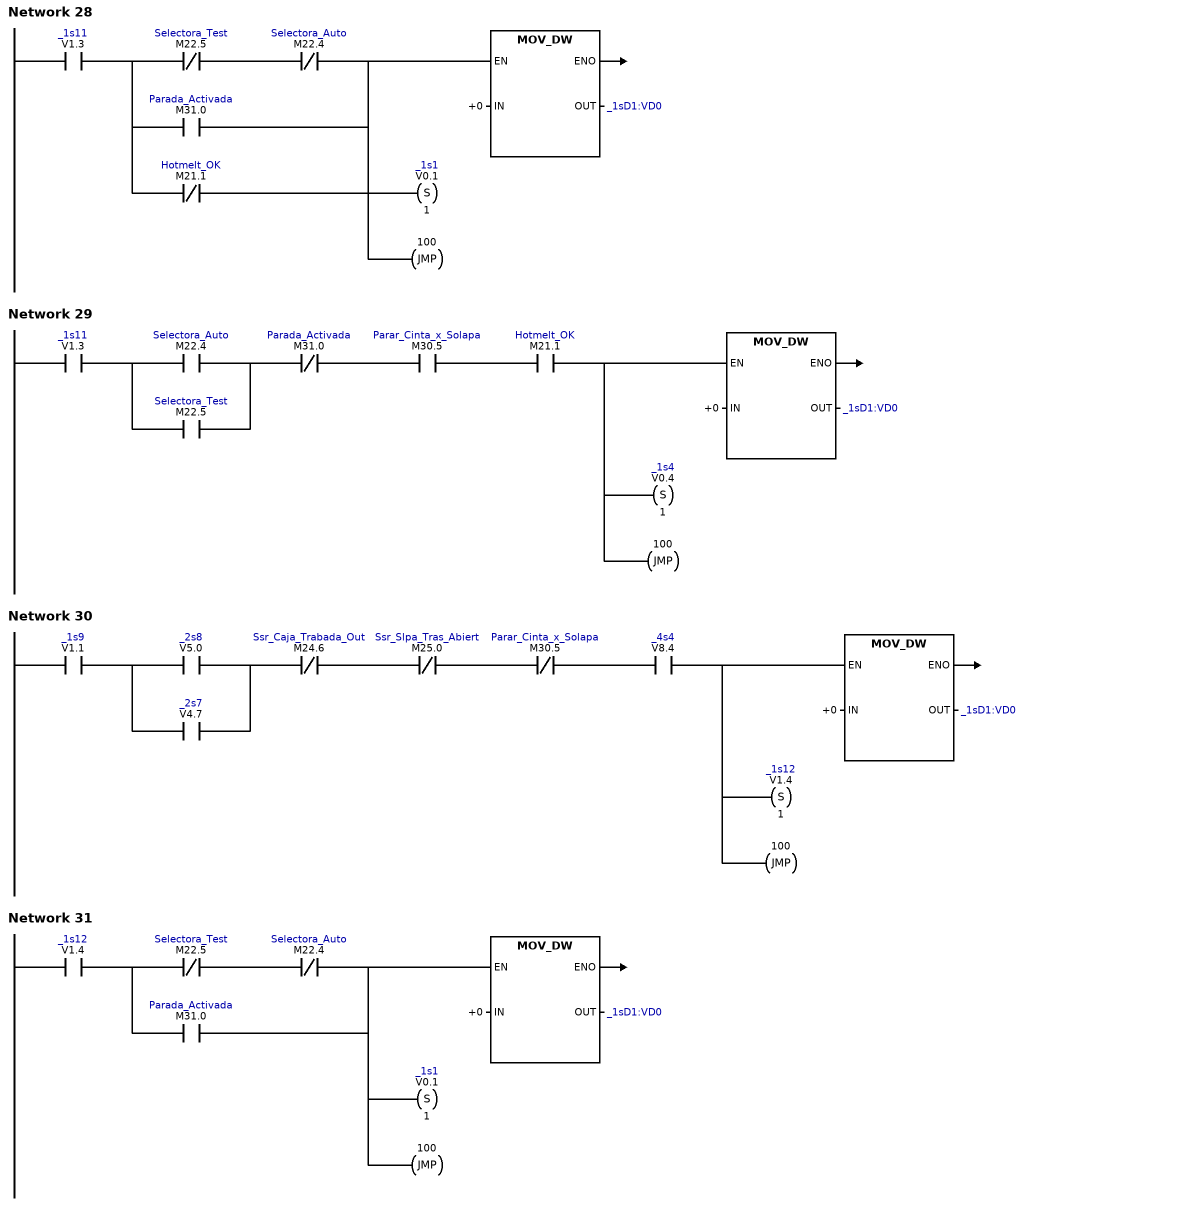
Network 28
LD     _1s11:V1.3
LDN    Selectora_Test:M22.5
AN     Selectora_Auto:M22.4
O      Parada_Activada:M31.0
ON     Hotmelt_OK:M21.1
ALD
MOVD   +0, _1sD1:VD0
S      _1s1:V0.1, 1
JMP    100
Network 29
LD     _1s11:V1.3
LD     Selectora_Auto:M22.4
O      Selectora_Test:M22.5
ALD
AN     Parada_Activada:M31.0
A      Parar_Cinta_x_Solapa:M30.5
A      Hotmelt_OK:M21.1
MOVD   +0, _1sD1:VD0
S      _1s4:V0.4, 1
JMP    100
Network 30
LD     _1s9:V1.1
LD     _2s8:V5.0
O      _2s7:V4.7
ALD
AN     Ssr_Caja_Trabada_Out:M24.6
AN     Ssr_Slpa_Tras_Abiert:M25.0
AN     Parar_Cinta_x_Solapa:M30.5
A      _4s4:V8.4
MOVD   +0, _1sD1:VD0
S      _1s12:V1.4, 1
JMP    100
Network 31
LD     _1s12:V1.4
LDN    Selectora_Test:M22.5
AN     Selectora_Auto:M22.4
O      Parada_Activada:M31.0
ALD
MOVD   +0, _1sD1:VD0
S      _1s1:V0.1, 1
JMP    100
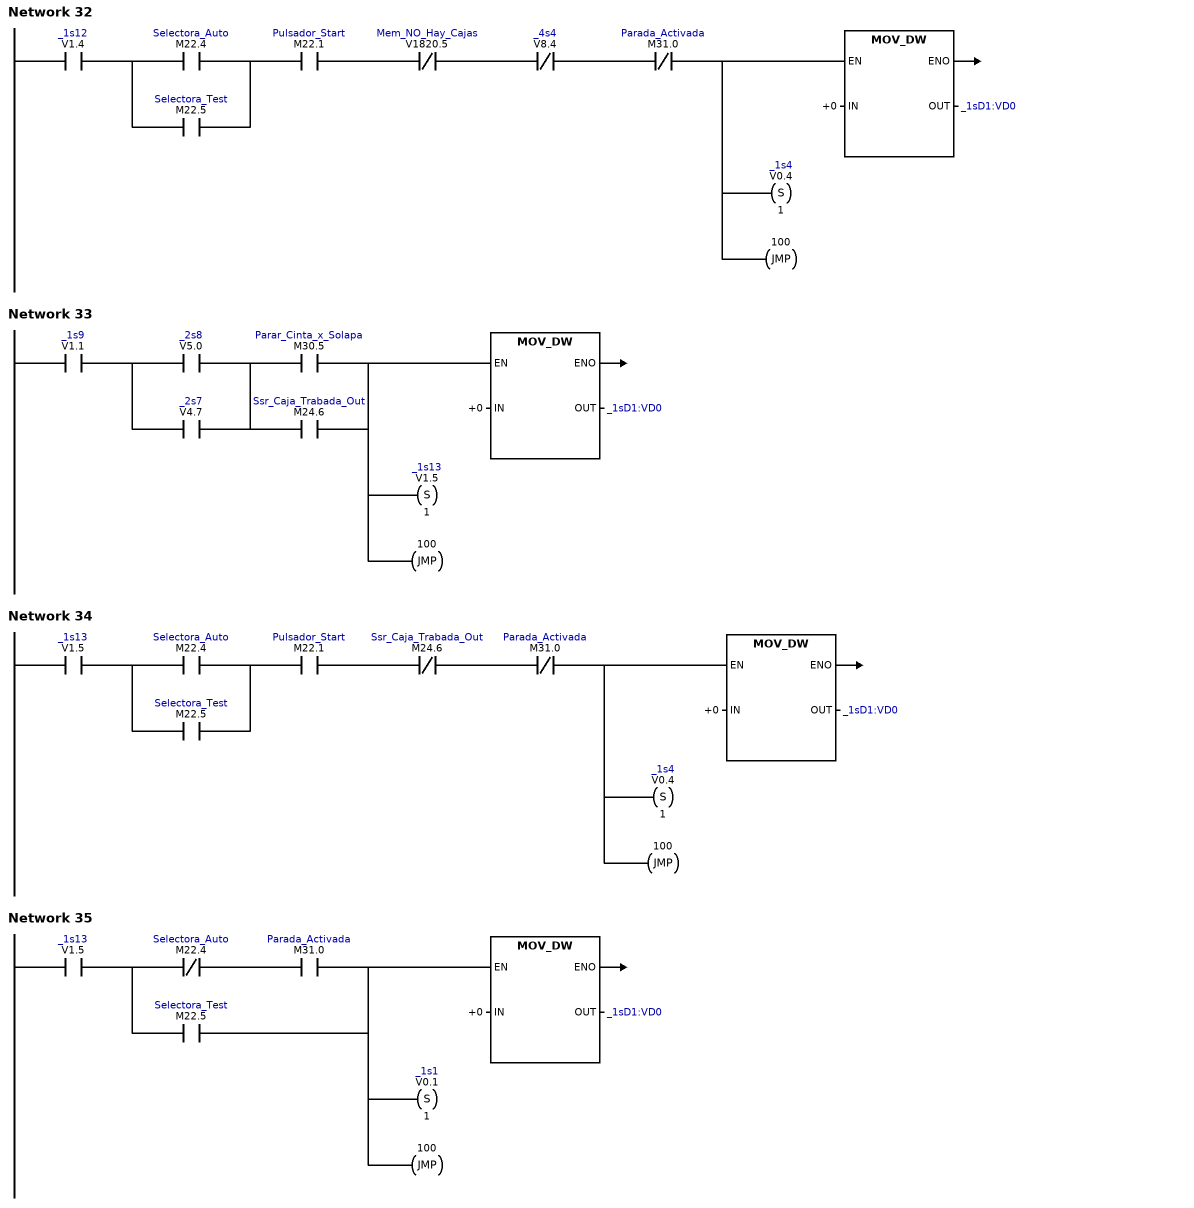
Network 32
LD     _1s12:V1.4
LD     Selectora_Auto:M22.4
O      Selectora_Test:M22.5
ALD
A      Pulsador_Start:M22.1
AN     Mem_NO_Hay_Cajas:V1820.5
AN     _4s4:V8.4
AN     Parada_Activada:M31.0
MOVD   +0, _1sD1:VD0
S      _1s4:V0.4, 1
JMP    100
Network 33
LD     _1s9:V1.1
LD     _2s8:V5.0
O      _2s7:V4.7
ALD
LD     Parar_Cinta_x_Solapa:M30.5
O      Ssr_Caja_Trabada_Out:M24.6
ALD
MOVD   +0, _1sD1:VD0
S      _1s13:V1.5, 1
JMP    100
Network 34
LD     _1s13:V1.5
LD     Selectora_Auto:M22.4
O      Selectora_Test:M22.5
ALD
A      Pulsador_Start:M22.1
AN     Ssr_Caja_Trabada_Out:M24.6
AN     Parada_Activada:M31.0
MOVD   +0, _1sD1:VD0
S      _1s4:V0.4, 1
JMP    100
Network 35
LD     _1s13:V1.5
LDN    Selectora_Auto:M22.4
A      Parada_Activada:M31.0
O      Selectora_Test:M22.5
ALD
MOVD   +0, _1sD1:VD0
S      _1s1:V0.1, 1
JMP    100
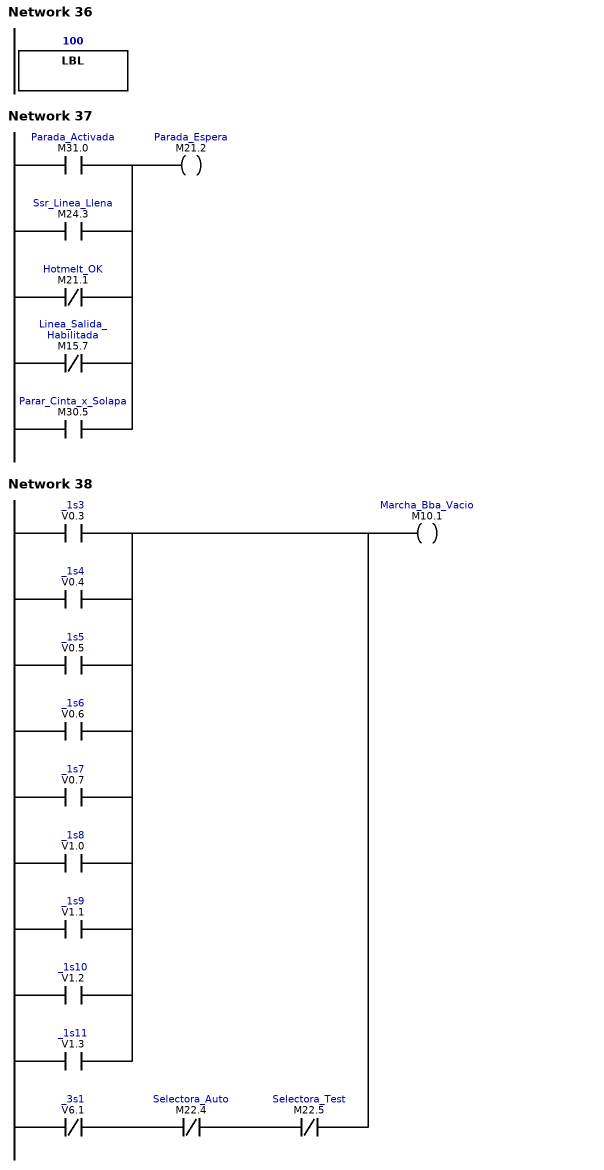
Network 36
LBL    100
Network 37
LD     Parada_Activada:M31.0
O      Ssr_Linea_Llena:M24.3
ON     Hotmelt_OK:M21.1
ON     Linea_Salida_Habilitada:M15.7
O      Parar_Cinta_x_Solapa:M30.5
=      Parada_Espera:M21.2
Network 38
LD     _1s3:V0.3
O      _1s4:V0.4
O      _1s5:V0.5
O      _1s6:V0.6
O      _1s7:V0.7
O      _1s8:V1.0
O      _1s9:V1.1
O      _1s10:V1.2
O      _1s11:V1.3
LDN    _3s1:V6.1
AN     Selectora_Auto:M22.4
AN     Selectora_Test:M22.5
OLD
=      Marcha_Bba_Vacio:M10.1
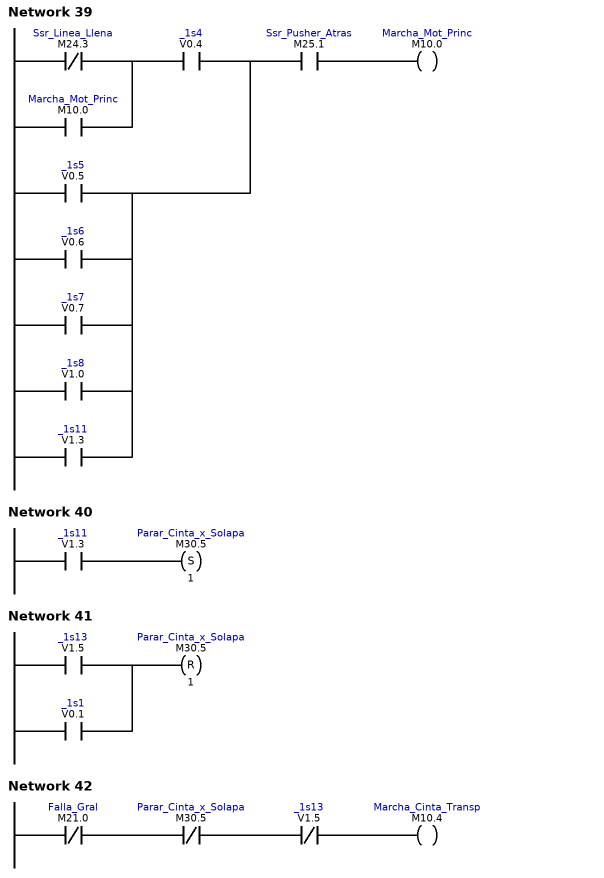
Network 39
LDN    Ssr_Linea_Llena:M24.3
O      Marcha_Mot_Princ:M10.0
A      _1s4:V0.4
LD     _1s5:V0.5
O      _1s6:V0.6
O      _1s7:V0.7
O      _1s8:V1.0
O      _1s11:V1.3
OLD
A      Ssr_Pusher_Atras:M25.1
=      Marcha_Mot_Princ:M10.0
Network 40
LD     _1s11:V1.3
S      Parar_Cinta_x_Solapa:M30.5, 1
Network 41
LD     _1s13:V1.5
O      _1s1:V0.1
R      Parar_Cinta_x_Solapa:M30.5, 1
Network 42
LDN    Falla_Gral:M21.0
AN     Parar_Cinta_x_Solapa:M30.5
AN     _1s13:V1.5
=      Marcha_Cinta_Transp:M10.4
